(* IEC 61131-3 sources: B-R/MBA, 12 files *)

(* ---- Main.st ---- *)
PROGRAM _INIT
	(* Insert code here *)
	MBAPid0510Para.set_value := 25;
	MBAPid0802Para.set_value := 30;
	MBAPid0510Para.gain := 400;
	MBAPid0802Para.gain := 60;
	MBAPid0510Para.integration_time := 45;
	MBAPid0802Para.integration_time := 240;
	MBAPid0510Para.derivative_time := 30;
	MBAPid0802Para.derivative_time := 0;

END_PROGRAM

PROGRAM _CYCLIC
	(* Insert code here *)
	S1A_ACT;
	S1B_ACT;
	S2_ACT;
	S3_ACT;
	S4_ACT;
	S5_ACT;
	S6_ACT;
	S7_ACT;
	S8_ACT;
	S9_ACT;
	S10_ACT;
END_PROGRAM

(* ---- MBAS10_ACTION.st ---- *)
ACTION S10_ACT:
	//设定时间
	FOR i := 0 TO MBAS10_STEP_NUM DO
		IF MBAS10_ST[i] < T#5s THEN
			MBAS10_ST[i] := T#5s;
		END_IF;
		MBAS10_STEP[i].set_time := MBAS10_ST[i];
	END_FOR;

	//流程步骤
	ProcessHandleFC(MBAS10,MBAS10_STEP[0],MBAS10_STEP_NUM);

	//object 手自动切换
	IF (MBAS10.status.mode <> 0) AND (NOT MBAS10.auto_mode_edge) THEN
		MBAS10.auto_mode_edge := TRUE;
		MBAS10.manual_mode_edge := FALSE;

		MBAR11.control.auto_operate := TRUE;
		MBAXV0811.control.auto_operate := TRUE;
		MBAXV0807.control.auto_operate := TRUE;
		MBAXV0808.control.auto_operate := TRUE;
		MBAXV0809.control.auto_operate := TRUE;
		MBAP09.control.auto_operate := TRUE;
		MBATV0801A.control.auto_operate := TRUE;
		MBATV0801B.control.auto_operate := TRUE;
		MBAXV0806.control.auto_operate := TRUE;
		MBAXV0812.control.auto_operate := TRUE;
		MBATVT0802.control.auto_operate := TRUE;
	END_IF;

	IF (MBAS10.status.mode = 0) AND (NOT MBAS10.manual_mode_edge) THEN
		MBAS10.manual_mode_edge := TRUE;
		MBAS10.auto_mode_edge := FALSE;

		MBAR11.control.manual_operate := TRUE;
		MBAXV0811.control.manual_operate := TRUE;
		MBAXV0807.control.manual_operate := TRUE;
		MBAXV0808.control.manual_operate := TRUE;
		MBAXV0809.control.manual_operate := TRUE;
		MBAP09.control.manual_operate := TRUE;
		MBATV0801A.control.manual_operate := TRUE;
		MBATV0801B.control.manual_operate := TRUE;
		MBAXV0806.control.manual_operate := TRUE;
		MBAXV0812.control.manual_operate := TRUE;
		MBATVT0802.control.manual_operate := TRUE;
	END_IF;

	//错误信号停机
	MBAS10.input.error_signal := (MBAR11.status.motor_status >= 2) OR (MBAXV0811.status.valve_status >= 2) OR
	(MBAXV0807.status.valve_status >= 2) OR (MBAXV0808.status.valve_status >= 2) OR (MBAXV0809.status.valve_status >= 2) OR
	(MBAP09.status.motor_status >= 2) OR (MBATV0801A.status.valve_status >= 2) OR (MBATV0801B.status.valve_status >= 2) OR
	(MBAXV0806.status.valve_status >= 2) OR (MBAXV0812.status.valve_status >= 2) OR (MBATVT0802.status.regulator_status >= 2);

	//MBAXV0814 玻璃塔出料自动
	SquareWave_0(open_time := DINT_TO_TIME(MBAXV0814_Open_Time * 1000), close_time := DINT_TO_TIME(MBAXV0814_Close_Time * 1000), on_off := TRUE, out := MBAXV0814.input.auto_open_signal);
	IF MBAS10.status.run_state = 1 THEN
		//步骤执行动作
		CASE MBAS10.status.run_step OF
			0:
				MBAS10_STEP[0].done := TRUE;
			1:
				//人工加料
			2:
				MBAR11.input.auto_run_signal := TRUE;
				MBAXV0811.input.auto_open_signal := TRUE;
				MBAXV0807.input.auto_open_signal := TRUE;
				MBAXV0808.input.auto_open_signal := TRUE;
				MBAXV0809.input.auto_open_signal := TRUE;
				MBAP09.input.auto_run_signal := TRUE;
				MTBasicsPID_1.Enable := TRUE;
				MBAS10_STEP[2].done := TRUE;
			3:
				IF (MBATIT0801.status.value < MBAS10_PARA_Temp1) AND (NOT MBAS10_STEP[3].done) THEN
	 				MBATV0801A.input.auto_open_signal := TRUE;
				END_IF;
				IF MBATIT0801.status.value >= MBAS10_PARA_Temp1 THEN
					MBATV0801B.input.auto_open_signal := TRUE;
					MBATV0801A.input.auto_open_signal := FALSE;
					MBAS10_STEP[3].done := TRUE;
				END_IF;
			4:

			5:
				IF MBATIT0803.status.value >= MBAS10_PARA_Temp2 THEN
					MBAXV0806.input.auto_open_signal := TRUE;
					MBAXV0807.input.auto_open_signal := FALSE;
					MBAXV0808.input.auto_open_signal := FALSE;
					MBAS10_STEP[5].done := TRUE;
				END_IF;
			6:
				IF MBATIT0801.status.value >= MBAS10_PARA_Temp3 THEN
					MBATV0801B.input.auto_open_signal := FALSE;
					MBAXV0807.input.auto_open_signal := TRUE;
					MBAXV0808.input.auto_open_signal := TRUE;
					MBAXV0806.input.auto_open_signal := FALSE;
					MBAXV0809.input.auto_open_signal := FALSE;
					MBAS10_STEP[6].done := TRUE;
				END_IF;
			7:
				IF MBATIT0801.status.value <= MBAS10_PARA_Temp4 THEN
					MBAXV0807.input.auto_open_signal := FALSE;
					MBAXV0808.input.auto_open_signal := FALSE;
					MBAXV0812.input.auto_open_signal := TRUE;
					MBAP09.input.auto_run_signal := FALSE;
					MBAS10_STEP[7].done := TRUE;
				END_IF;
			8:
			//人工操作
		END_CASE;
	END_IF;

	//TSV0510调节
	R_TRIG_3(CLK := MBATVT0802.status.auto_mode);
	IF R_TRIG_3.Q THEN
		MTBasicsPID_1.Enable := TRUE;
	END_IF;
	F_TRIG_3(CLK := MBATVT0802.status.auto_mode);
	IF F_TRIG_3.Q THEN
		MTBasicsPID_1.Enable := FALSE;
	END_IF;
	//MTBasicsPID_1.Enable := TRUE;
	MTBasicsPID_1.Invert := TRUE;
	MTBasicsPID_1.PIDParameters.Gain := MBAPid0802Para.gain;
	MTBasicsPID_1.PIDParameters.DerivativeTime := MBAPid0802Para.derivative_time;
	MTBasicsPID_1.PIDParameters.IntegrationTime := MBAPid0802Para.integration_time;
	MTBasicsPID_1.MinOut := 0.0;
	MTBasicsPID_1.MaxOut := 100.0;
	MTBasicsPID_1.SetValue := MBAPid0802Para.set_value;
	MTBasicsPID_1.ActValue := MBATIT0802.status.value;
	MTBasicsPID_1.Update := MBAPid0802.update;
	MTBasicsPID_1();
	MBAPid0802.out := MTBasicsPID_1.Out;
	IF MTBasicsPID_1.Active THEN
		MBATVT0802.input.auto_degree_set := MTBasicsPID_1.Out;
	ELSE
		MBATVT0802.input.auto_degree_set := 0.0;
	END_IF;
	IF MTBasicsPID_1.UpdateDone THEN
		MBAPid0802.update := FALSE;
	END_IF;

	//人工确认步骤可用
	IF (MBAS10.status.run_state) AND (NOT MBAS10_STEP[MBAS10.status.run_step].done AND ((MBAS10.status.run_step = 1) OR (MBAS10.status.run_step = 4) OR (MBAS10.status.run_step = 8))) THEN
		MBAS10.status.confirm_enable := TRUE;
	ELSE
		MBAS10.status.confirm_enable := FALSE;
	END_IF;
END_ACTION

(* ---- MBAS1A_ACTION.st ---- *)
ACTION S1A_ACT:
	//设定时间
	FOR i := 0 TO MBAS1_STEP_NUM DO
		IF MBAS1A_ST[i] < T#5s THEN
			MBAS1A_ST[i] := T#5s;
		END_IF;
		MBAS1A_STEP[i].set_time := MBAS1A_ST[i];
	END_FOR;

	//流程步骤
	ProcessHandleFC(MBAS1A,MBAS1A_STEP[0],MBAS1_STEP_NUM);

	//object 手自动切换
	IF (MBAS1A.status.mode <> 0) AND (NOT MBAS1A.auto_mode_edge) THEN
		MBAS1A.auto_mode_edge := TRUE;
		MBAS1A.manual_mode_edge := FALSE;

		STFLV0101.control.auto_operate := TRUE;
		STFLV0102.control.auto_operate := TRUE;
		MBALV0102.control.auto_operate := TRUE;
		STFP01.control.auto_operate := TRUE;
		STFLV3601.control.auto_operate := TRUE;
		STFLV3602.control.auto_operate := TRUE;
		MBALV0103.control.auto_operate := TRUE;
		STFP36.control.auto_operate := TRUE;
		MBALV0101.control.auto_operate := TRUE;
		MBAXV0105.control.auto_operate := TRUE;
		MBAXV0103.control.auto_operate := TRUE;
		MBAAV0101A.control.auto_operate := TRUE;
		MBAR01A.control.auto_operate := TRUE;
		MBAXV0102.control.auto_operate := TRUE;
		MBAXV0101.control.auto_operate := TRUE;
		MBAAV0101B.control.auto_operate := TRUE;
		MBAXV0209.control.auto_operate := TRUE;
		MBAXV0212.control.auto_operate := TRUE;
		MBAXV0104.control.auto_operate := TRUE;
		MBAXV0415.control.auto_operate := TRUE;
	END_IF;

	IF (MBAS1A.status.mode = 0) AND (NOT MBAS1A.manual_mode_edge) THEN
		MBAS1A.manual_mode_edge := TRUE;
		MBAS1A.auto_mode_edge := FALSE;

		STFLV0101.control.manual_operate := TRUE;
		STFLV0102.control.manual_operate := TRUE;
		MBALV0102.control.manual_operate := TRUE;
		STFP01.control.manual_operate := TRUE;
		STFLV3601.control.manual_operate := TRUE;
		STFLV3602.control.manual_operate := TRUE;
		MBALV0103.control.manual_operate := TRUE;
		STFP36.control.manual_operate := TRUE;
		MBALV0101.control.manual_operate := TRUE;
		MBAXV0105.control.manual_operate := TRUE;
		MBAXV0103.control.manual_operate := TRUE;
		MBAAV0101A.control.manual_operate := TRUE;
		MBAR01A.control.manual_operate := TRUE;
		MBAXV0102.control.manual_operate := TRUE;
		MBAXV0101.control.manual_operate := TRUE;
		MBAAV0101B.control.manual_operate := TRUE;
		MBAXV0209.control.manual_operate := TRUE;
		MBAXV0212.control.manual_operate := TRUE;
		MBAXV0104.control.manual_operate := TRUE;
		MBAXV0415.control.manual_operate := TRUE;
	END_IF;

	//错误信号停机
	MBAS1A.input.error_signal := (STFLV0101.status.valve_status >= 2) OR (STFLV0102.status.valve_status >= 2) OR
	(MBALV0102.status.valve_status >= 2) OR (STFP01.status.motor_status >= 2) OR (STFLV3601.status.valve_status >= 2) OR
	(STFLV3602.status.valve_status >= 2) OR (MBALV0103.status.valve_status >= 2) OR (STFP36.status.motor_status >= 2) OR
	(MBALV0101.status.valve_status >= 2) OR (MBAXV0105.status.valve_status >= 2) OR (MBAXV0103.status.valve_status >= 2) OR
	(MBAAV0101A.status.valve_status >= 2) OR (MBAR01A.status.motor_status >= 2) OR (MBAXV0102.status.valve_status >= 2) OR
	(MBAXV0101.status.valve_status >= 2) OR (MBAAV0101B.status.valve_status >= 2) OR (MBAXV0209.status.valve_status >= 2) OR
	(MBAXV0212.status.valve_status >= 2) OR (MBAXV0104.status.valve_status >= 2) OR (MBAXV0415.status.valve_status >= 2);

	IF MBAS1A.status.run_state = 1 THEN
		//步骤执行动作
		CASE MBAS1A.status.run_step OF
			0:
				IF NOT MBAS1A_STEP[0].done  THEN
					STFLV0101.control.auto_operate := TRUE;
					STFLV0102.control.auto_operate := TRUE;
					MBALV0104.control.auto_operate := TRUE;
					STFP01.control.auto_operate := TRUE;
					STFLV3601.control.auto_operate := TRUE;
					STFLV3602.control.auto_operate := TRUE;
					MBALV0105.control.auto_operate := TRUE;
					STFP36.control.auto_operate := TRUE;
					MBALV0101.control.auto_operate := TRUE;
					MBAXV0110.control.auto_operate := TRUE;
					MBAXV0108.control.auto_operate := TRUE;
					MBAAV0102A.control.auto_operate := TRUE;
					MBAR01B.control.auto_operate := TRUE;
					MBAXV0107.control.auto_operate := TRUE;
					MBAXV0106.control.auto_operate := TRUE;
					MBAAV0102B.control.auto_operate := TRUE;
					MBAXV0209.control.auto_operate := TRUE;
					MBAXV0212.control.auto_operate := TRUE;
					MBAXV0109.control.auto_operate := TRUE;
					MBAXV0415.control.auto_operate := TRUE;
					MBAS1A_STEP[0].done := TRUE;
				END_IF;
			1:
				//高位槽进料
			2:
				CASE step1_4a OF
					0:
						IF NOT MBAS1A_STEP[2].done THEN
							step1_4a := 1;
						END_IF;
					1:
						MBAXV0105.input.auto_open_signal := TRUE;
						step1_4a := 2;
					2:
						TON_8.PT := DINT_TO_TIME(MBAS1A_PARA_T4 * 1000);
						TON_8.IN := TRUE;
						IF TON_8.Q THEN
							TON_8.IN := FALSE;
							step1_4a := 3;
						END_IF;
					3:
						MBAXV0105.input.auto_open_signal := FALSE;
						step1_4a := 4;
					4:
						MBAXV0103.input.auto_open_signal := TRUE;
						IF MBAXV0103.input.open_feedback_state THEN
							step1_4a := 5;
						END_IF;
					5:
						IF MBALIT0101.status.value <= MBAS1A_PARA_L4 THEN
							step1_4a := 6;
						END_IF;
					6:
						TON_8.PT := DINT_TO_TIME(MBAS1A_PARA_T5 * 60 * 1000);
						TON_8.IN := TRUE;
						IF TON_8.Q THEN
							TON_8.IN := FALSE;
							step1_4a := 7;
						END_IF;
					7:
						MBAXV0103.input.auto_open_signal := FALSE;
						IF MBAXV0103.input.close_feedback_state THEN
							step1_4a := 0;
							MBAS1A_STEP[2].done := TRUE;
						END_IF;
				END_CASE;
				TON_8();
			3:
				//人工投料,结束后确认
			4:
				CASE step1_6a OF
					0:
						IF NOT MBAS1A_STEP[4].done THEN
							step1_6a := 1;
						END_IF;
					1:
						LiquidRelease_3(sp_time := DINT_TO_TIME(MBAS1A_PARA_T10 * 60 * 1000),
						level_value := MBALIT0102.status.value,
						set_point := MBAS1A_PARA_L5,
						done := step1_6a_1_done);
						MBAAV0101A.input.auto_open_signal := LiquidRelease_3.run;
						IF step1_6a_1_done AND MBAAV0101A.input.close_feedback_state AND (NOT MBAAV0101A.input.auto_open_signal) THEN
							step1_6a := 2;
						END_IF;
					2:
						MBAR01A.input.auto_run_signal := TRUE;
						IF MBAR01A.input.run_feedback THEN
							step1_6a := 0;
							step1_6a_1_done := FALSE;
							MBAS1A_STEP[4].done := TRUE;
						END_IF;
				END_CASE;
			5:
				CASE step1_7a OF
					0:
						IF NOT MBAS1A_STEP[5].done THEN
							step1_7a := 1;
						END_IF;
					1:
						TON_13.PT := DINT_TO_TIME(MBAS1A_PARA_T6 * 60 * 1000);
						TON_13.IN := TRUE;
						IF TON_13.Q THEN
							TON_13.IN := FALSE;
							step1_7a := 2;
						END_IF;
					2:
						MBAXV0101.input.auto_open_signal := TRUE;
						IF MBAXV0101.input.open_feedback_state THEN
							step1_7a := 3;
						END_IF;
					3:
						IF MBATIT0101.status.value >= MBAS1A_PARA_Temp1 THEN
							step1_7a := 4;
						END_IF;
					4:
						MBAXV0102.input.auto_open_signal := TRUE;
						IF MBAXV0102.input.open_feedback_state THEN
							step1_7a := 5;
						END_IF;
					5:
						TON_13.PT := DINT_TO_TIME(MBAS1A_PARA_T7 * 60 * 1000);
						TON_13.IN := TRUE;
						IF TON_13.Q THEN
							TON_13.IN := FALSE;
							step1_7a := 6;
						END_IF;
					6:
						MBAAV0101B.input.auto_open_signal := TRUE;
						IF MBAAV0101B.input.open_feedback_state THEN
							step1_7a := 7;
						END_IF;
					7:
						TON_13.PT := DINT_TO_TIME(MBAS1A_PARA_T8 * 60 * 1000);
						TON_13.IN := TRUE;
						IF TON_13.Q THEN
							TON_13.IN := FALSE;
							step1_7a := 8;
						END_IF;
					8:
						MBAAV0101A.input.auto_open_signal := TRUE;
						IF MBAAV0101A.input.open_feedback_state THEN
							step1_7a := 9;
						END_IF;
					9:
						TON_13.PT := DINT_TO_TIME(MBAS1A_PARA_T9 * 60 * 1000);
						TON_13.IN := TRUE;
						IF TON_13.Q THEN
							TON_13.IN := FALSE;
							step1_7a := 10;
						END_IF;
					10:
						MBAXV0102.input.auto_open_signal := FALSE;
						MBAAV0101A.input.auto_open_signal := FALSE;
						MBAAV0101B.input.auto_open_signal := FALSE;
						IF MBAXV0102.input.close_feedback_state AND MBAAV0101A.input.close_feedback_state AND MBAAV0101B.input.close_feedback_state THEN
							step1_7a := 0;
							MBAS1A_STEP[5].done := TRUE;
						END_IF;
				END_CASE;
				TON_13();
			6:
				//人工确认MBAR13空闲
			7:
				MBAXV0209.input.auto_open_signal := TRUE;
				MBAXV0212.input.auto_open_signal := TRUE;
				MBAXV0415.input.auto_open_signal := TRUE;
				IF MBAXV0209.input.open_feedback_state AND MBAXV0212.input.open_feedback_state AND MBAXV0415.input.open_feedback_state THEN
					MBAXV0104.input.auto_open_signal := TRUE;
					MBAR01A.input.auto_run_signal := FALSE;
				END_IF;
				IF MBAXV0209.input.open_feedback_state AND MBAXV0212.input.open_feedback_state AND MBAXV0415.input.open_feedback_state AND MBAXV0104.input.open_feedback_state AND (NOT MBAR01A.input.run_feedback) THEN
					MBAS1A_STEP[7].done := TRUE;
				END_IF;
			8:
				//人工确认转移完毕
			9:
				MBAXV0104.input.auto_open_signal := FALSE;
				MBAXV0101.input.auto_open_signal := FALSE;
				IF MBAXV0104.input.close_feedback_state AND MBAXV0101.input.close_feedback_state THEN
					MBAS1A_STEP[9].done := TRUE;
				END_IF;
		END_CASE;
	END_IF;

	IF mba_v02a_add THEN
		CASE step1_1a OF
			0:
				step1_1a := 1;
			1:
				STFLV0101.input.auto_open_signal := FALSE;
				STFLV0102.input.auto_open_signal := FALSE;
				MBALV0102.input.auto_open_signal := TRUE;
				IF STFLV0102.input.close_feedback_state AND STFLV0101.input.close_feedback_state AND MBALV0102.input.open_feedback_state THEN
					step1_1a := 2;
				END_IF;
			2:
				LiquidAdd_0(level_value := MBALIT0102.status.value,
				sp_value := MBAS1A_PARA_L1,
				sp_accumulation := MBAS1A_PARA_AC1,
				sp_time := DINT_TO_TIME(MBAS1A_PARA_T1 * 1000),
				flowmeter := STFFQIT0102,
				done := step1_1a_2_done);
				STFP01.input.auto_run_signal := LiquidAdd_0.run;
				IF step1_1a_2_done AND (NOT STFP01.input.run_feedback) AND (NOT STFP01.input.auto_run_signal) THEN
					step1_1a := 3;
				END_IF;
			3:
				IF STFFQIT0102.flowrate <= flowrate_threshold THEN
					step1_1a := 4;
				END_IF;
			4:
				MBALV0102.input.auto_open_signal := FALSE;
				IF MBALV0102.input.close_feedback_state THEN
					step1_1a_2_done := FALSE;
					step1_1a := 0;
					mba_v02a_add := FALSE;
				END_IF;
		END_CASE;
	END_IF;

	IF mba_v03a_add THEN
		CASE step1_2a OF
			0:
				step1_2a := 1;
			1:
				STFLV3601.input.auto_open_signal := TRUE;
				STFLV3602.input.auto_open_signal := FALSE;
				MBALV0103.input.auto_open_signal := TRUE;
				IF STFLV3601.input.open_feedback_state AND STFLV3602.input.close_feedback_state AND MBALV0103.input.open_feedback_state THEN
					step1_2a := 2;
				END_IF;
			2:
				LiquidAdd_1(level_value := MBALIT0103.status.value,
				sp_value := MBAS1A_PARA_L2,
				sp_accumulation := MBAS1A_PARA_AC2,
				sp_time := DINT_TO_TIME(MBAS1A_PARA_T2 * 1000),
				flowmeter := STFFQIT3602,
				done := step1_2a_2_done);
				STFP36.input.auto_run_signal := LiquidAdd_1.run;
				IF step1_2a_2_done AND (NOT STFP36.input.run_feedback) AND (NOT STFP36.input.auto_run_signal) THEN
					step1_2a := 3;
				END_IF;
			3:
				IF STFFQIT3602.flowrate <= flowrate_threshold THEN
					step1_2a := 4;
				END_IF;
			4:
				MBALV0103.input.auto_open_signal := FALSE;
				IF MBALV0103.input.close_feedback_state THEN
					step1_2a := 0;
					step1_2a_2_done := FALSE;
					mba_v03a_add := FALSE;
				END_IF;
		END_CASE;
	END_IF;

	//人工确认步骤可用
	IF (MBAS1A.status.run_state) AND (NOT MBAS1A_STEP[MBAS1A.status.run_step].done AND ((MBAS1A.status.run_step = 1) OR (MBAS1A.status.run_step = 3) OR (MBAS1A.status.run_step = 6) OR (MBAS1A.status.run_step = 8))) THEN
		MBAS1A.status.confirm_enable := TRUE;
	ELSE
		MBAS1A.status.confirm_enable := FALSE;
	END_IF;
END_ACTION

(* ---- MBAS1B_ACTION.st ---- *)
ACTION S1B_ACT:
	//设定时间
	FOR i := 0 TO MBAS1_STEP_NUM DO
		IF MBAS1B_ST[i] < T#5s THEN
			MBAS1B_ST[i] := T#5s;
		END_IF;
		MBAS1B_STEP[i].set_time := MBAS1B_ST[i];
	END_FOR;

	//流程步骤
	ProcessHandleFC(MBAS1B,MBAS1B_STEP[0],MBAS1_STEP_NUM);

	//object 手自动切换
	IF (MBAS1B.status.mode <> 0) AND (NOT MBAS1B.auto_mode_edge) THEN
		MBAS1B.auto_mode_edge := TRUE;
		MBAS1B.manual_mode_edge := FALSE;

		STFLV0101.control.auto_operate := TRUE;
		STFLV0102.control.auto_operate := TRUE;
		MBALV0104.control.auto_operate := TRUE;
		STFP01.control.auto_operate := TRUE;
		STFLV3601.control.auto_operate := TRUE;
		STFLV3602.control.auto_operate := TRUE;
		MBALV0105.control.auto_operate := TRUE;
		STFP36.control.auto_operate := TRUE;
		MBALV0101.control.auto_operate := TRUE;
		MBAXV0110.control.auto_operate := TRUE;
		MBAXV0108.control.auto_operate := TRUE;
		MBAAV0102A.control.auto_operate := TRUE;
		MBAR01B.control.auto_operate := TRUE;
		MBAXV0107.control.auto_operate := TRUE;
		MBAXV0106.control.auto_operate := TRUE;
		MBAAV0102B.control.auto_operate := TRUE;
		MBAXV0209.control.auto_operate := TRUE;
		MBAXV0212.control.auto_operate := TRUE;
		MBAXV0109.control.auto_operate := TRUE;
		MBAXV0415.control.auto_operate := TRUE;
	END_IF;

	IF (MBAS1B.status.mode = 0) AND (NOT MBAS1B.manual_mode_edge) THEN
		MBAS1B.manual_mode_edge := TRUE;
		MBAS1B.auto_mode_edge := FALSE;

		STFLV0101.control.manual_operate := TRUE;
		STFLV0102.control.manual_operate := TRUE;
		MBALV0104.control.manual_operate := TRUE;
		STFP01.control.manual_operate := TRUE;
		STFLV3601.control.manual_operate := TRUE;
		STFLV3602.control.manual_operate := TRUE;
		MBALV0105.control.manual_operate := TRUE;
		STFP36.control.manual_operate := TRUE;
		MBALV0101.control.manual_operate := TRUE;
		MBAXV0110.control.manual_operate := TRUE;
		MBAXV0108.control.manual_operate := TRUE;
		MBAAV0102A.control.manual_operate := TRUE;
		MBAR01B.control.manual_operate := TRUE;
		MBAXV0107.control.manual_operate := TRUE;
		MBAXV0106.control.manual_operate := TRUE;
		MBAAV0102B.control.manual_operate := TRUE;
		MBAXV0209.control.manual_operate := TRUE;
		MBAXV0212.control.manual_operate := TRUE;
		MBAXV0109.control.manual_operate := TRUE;
		MBAXV0415.control.manual_operate := TRUE;
	END_IF;

	//错误信号停机
	MBAS1B.input.error_signal := (STFLV0101.status.valve_status >= 2) OR (STFLV0102.status.valve_status >= 2) OR
	(MBALV0104.status.valve_status >= 2) OR (STFP01.status.motor_status >= 2) OR (STFLV3601.status.valve_status >= 2) OR
	(STFLV3602.status.valve_status >= 2) OR (MBALV0105.status.valve_status >= 2) OR (STFP36.status.motor_status >= 2) OR
	(MBALV0101.status.valve_status >= 2) OR (MBAXV0110.status.valve_status >= 2) OR (MBAXV0108.status.valve_status >= 2) OR
	(MBAAV0102A.status.valve_status >= 2) OR (MBAR01B.status.motor_status >= 2) OR (MBAXV0107.status.valve_status >= 2) OR
	(MBAXV0106.status.valve_status >= 2) OR (MBAAV0102B.status.valve_status >= 2) OR (MBAXV0209.status.valve_status >= 2) OR
	(MBAXV0212.status.valve_status >= 2) OR (MBAXV0109.status.valve_status >= 2) OR (MBAXV0415.status.valve_status >= 2);

	IF MBAS1B.status.run_state = 1 THEN
		//步骤执行动作
		CASE MBAS1B.status.run_step OF
			0:
				IF NOT MBAS1B_STEP[0].done THEN
					STFLV0101.control.auto_operate := TRUE;
					STFLV0102.control.auto_operate := TRUE;
					MBALV0104.control.auto_operate := TRUE;
					STFP01.control.auto_operate := TRUE;
					STFLV3601.control.auto_operate := TRUE;
					STFLV3602.control.auto_operate := TRUE;
					MBALV0105.control.auto_operate := TRUE;
					STFP36.control.auto_operate := TRUE;
					MBALV0101.control.auto_operate := TRUE;
					MBAXV0110.control.auto_operate := TRUE;
					MBAXV0108.control.auto_operate := TRUE;
					MBAAV0102A.control.auto_operate := TRUE;
					MBAR01B.control.auto_operate := TRUE;
					MBAXV0107.control.auto_operate := TRUE;
					MBAXV0106.control.auto_operate := TRUE;
					MBAAV0102B.control.auto_operate := TRUE;
					MBAXV0209.control.auto_operate := TRUE;
					MBAXV0212.control.auto_operate := TRUE;
					MBAXV0109.control.auto_operate := TRUE;
					MBAXV0415.control.auto_operate := TRUE;
					MBAS1B_STEP[0].done := TRUE;
				END_IF;
			1:
				//高位槽进料
			2:
				CASE step1_4b OF
					0:
						IF NOT MBAS1B_STEP[2].done THEN
							step1_4b := 1;
						END_IF;
					1:
						MBAXV0110.input.auto_open_signal := TRUE;
						step1_4b := 2;
					2:
						TON_14.PT := DINT_TO_TIME(MBAS1B_PARA_T4 * 1000);
						TON_14.IN := TRUE;
						IF TON_14.Q THEN
							TON_14.IN := FALSE;
							step1_4b := 3;
						END_IF;
					3:
						MBAXV0110.input.auto_open_signal := FALSE;
						step1_4b := 4;
					4:
						MBAXV0108.input.auto_open_signal := TRUE;
						IF MBAXV0108.input.open_feedback_state THEN
							step1_4b := 5;
						END_IF;
					5:
						IF MBALIT0101.status.value <= MBAS1B_PARA_L4 THEN
							step1_4b := 6;
						END_IF;
					6:
						TON_14.PT := DINT_TO_TIME(MBAS1B_PARA_T5 * 60 * 1000);
						TON_14.IN := TRUE;
						IF TON_14.Q THEN
							TON_14.IN := FALSE;
							step1_4b := 7;
						END_IF;
					7:
						MBAXV0108.input.auto_open_signal := FALSE;
						IF MBAXV0108.input.close_feedback_state THEN
							step1_4b := 0;
							MBAS1B_STEP[2].done := TRUE;
						END_IF;
				END_CASE;
				TON_14();
			3:
				//人工投料,结束后确认
			4:
				CASE step1_6b OF
					0:
						IF NOT MBAS1B_STEP[4].done THEN
							step1_6b := 1;
						END_IF;
					1:
						LiquidRelease_1(sp_time := DINT_TO_TIME(MBAS1B_PARA_T10 * 60 * 1000),
						level_value := MBALIT0104.status.value,
						set_point := MBAS1B_PARA_L5,
						done := step1_6b_1_done);
						MBAAV0102A.input.auto_open_signal := LiquidRelease_1.run;
						IF step1_6b_1_done AND MBAAV0102A.input.close_feedback_state AND (NOT MBAAV0102A.input.auto_open_signal) THEN
							step1_6b := 2;
						END_IF;
					2:
						MBAR01B.input.auto_run_signal := TRUE;
						IF MBAR01B.input.run_feedback THEN
							step1_6b := 0;
							step1_6b_1_done := FALSE;
							MBAS1B_STEP[4].done := TRUE;
						END_IF;
				END_CASE;
			5:
				CASE step1_7b OF
					0:
						IF NOT MBAS1B_STEP[5].done THEN
							step1_7b := 1;
						END_IF;
					1:
						TON_15.PT := DINT_TO_TIME(MBAS1B_PARA_T6 * 60 * 1000);
						TON_15.IN := TRUE;
						IF TON_15.Q THEN
							TON_15.IN := FALSE;
							step1_7b := 2;
						END_IF;
					2:
						MBAXV0106.input.auto_open_signal := TRUE;
						IF MBAXV0106.input.open_feedback_state THEN
							step1_7b := 3;
						END_IF;
					3:
						IF MBATIT0102.status.value >= MBAS1B_PARA_Temp1 THEN
							step1_7b := 4;
						END_IF;
					4:
						MBAXV0107.input.auto_open_signal := TRUE;
						IF MBAXV0107.input.open_feedback_state THEN
							step1_7b := 5;
						END_IF;
					5:
						TON_15.PT := DINT_TO_TIME(MBAS1B_PARA_T7 * 60 * 1000);
						TON_15.IN := TRUE;
						IF TON_15.Q THEN
							TON_15.IN := FALSE;
							step1_7b := 6;
						END_IF;
					6:
						MBAAV0102B.input.auto_open_signal := TRUE;
						IF MBAAV0102B.input.open_feedback_state THEN
							step1_7b := 7;
						END_IF;
					7:
						TON_15.PT := DINT_TO_TIME(MBAS1B_PARA_T8 * 60 * 1000);
						TON_15.IN := TRUE;
						IF TON_15.Q THEN
							TON_15.IN := FALSE;
							step1_7b := 8;
						END_IF;
					8:
						MBAAV0102A.input.auto_open_signal := TRUE;
						IF MBAAV0102A.input.open_feedback_state THEN
							step1_7b := 9;
						END_IF;
					9:
						TON_15.PT := DINT_TO_TIME(MBAS1B_PARA_T9 * 60 * 1000);
						TON_15.IN := TRUE;
						IF TON_15.Q THEN
							TON_15.IN := FALSE;
							step1_7b := 10;
						END_IF;
					10:
						MBAXV0107.input.auto_open_signal := FALSE;
						MBAAV0102A.input.auto_open_signal := FALSE;
						MBAAV0102B.input.auto_open_signal := FALSE;
						IF MBAXV0107.input.close_feedback_state AND MBAAV0102A.input.close_feedback_state AND MBAAV0102B.input.close_feedback_state THEN
							step1_7b := 0;
							MBAS1B_STEP[5].done := TRUE;
						END_IF;
				END_CASE;
				TON_15();
			6:
				//人工确认MBAR13空闲
			7:
				MBAXV0209.input.auto_open_signal := TRUE;
				MBAXV0212.input.auto_open_signal := TRUE;
				MBAXV0415.input.auto_open_signal := TRUE;
				IF MBAXV0209.input.open_feedback_state AND MBAXV0212.input.open_feedback_state AND MBAXV0415.input.open_feedback_state THEN
					MBAXV0109.input.auto_open_signal := TRUE;
					MBAR01B.input.auto_run_signal := FALSE;
				END_IF;
				IF MBAXV0209.input.open_feedback_state AND MBAXV0212.input.open_feedback_state AND MBAXV0415.input.open_feedback_state AND MBAXV0109.input.open_feedback_state AND (NOT MBAR01B.input.run_feedback) THEN
					MBAS1B_STEP[7].done := TRUE;
				END_IF;
			8:
				//人工确认转移完毕
			9:
				MBAXV0109.input.auto_open_signal := FALSE;
				MBAXV0106.input.auto_open_signal := FALSE;
				IF MBAXV0109.input.close_feedback_state AND MBAXV0106.input.close_feedback_state THEN
					MBAS1B_STEP[9].done := TRUE;
				END_IF;
		END_CASE;
	END_IF;

	IF mba_v02b_add THEN
		CASE step1_1b OF
			0:
				step1_1b := 1;
			1:
				STFLV0101.input.auto_open_signal := FALSE;
				STFLV0102.input.auto_open_signal := FALSE;
				MBALV0104.input.auto_open_signal := TRUE;
				IF STFLV0102.input.close_feedback_state AND STFLV0101.input.close_feedback_state AND MBALV0104.input.open_feedback_state THEN
					step1_1b := 2;
				END_IF;
			2:
				LiquidAdd_4(level_value := MBALIT0104.status.value,
				sp_value := MBAS1B_PARA_L1,
				sp_accumulation := MBAS1B_PARA_AC1,
				sp_time := DINT_TO_TIME(MBAS1B_PARA_T1 * 1000),
				flowmeter := STFFQIT0102,
				done := step1_1b_2_done);
				STFP01.input.auto_run_signal := LiquidAdd_4.run;
				IF step1_1b_2_done AND (NOT STFP01.input.run_feedback) AND (NOT STFP01.input.auto_run_signal) THEN
					step1_1b := 3;
				END_IF;
			3:
				IF STFFQIT0102.flowrate <= flowrate_threshold THEN
					step1_1b := 4;
				END_IF;
			4:
				MBALV0104.input.auto_open_signal := FALSE;
				IF MBALV0104.input.close_feedback_state THEN
					step1_1b := 0;
					step1_1b_2_done := FALSE;
					mba_v02b_add := FALSE;
				END_IF;
		END_CASE;
	END_IF;

	IF mba_v03b_add THEN
		CASE step1_2b OF
			0:
				step1_2b := 1;
			1:
				STFLV3601.input.auto_open_signal := TRUE;
				STFLV3602.input.auto_open_signal := FALSE;
				MBALV0105.input.auto_open_signal := TRUE;
				IF STFLV3601.input.open_feedback_state AND STFLV3602.input.close_feedback_state AND MBALV0105.input.open_feedback_state THEN
					step1_2b := 2;
				END_IF;
			2:
				LiquidAdd_5(level_value := MBALIT0105.status.value,
				sp_value := MBAS1B_PARA_L2,
				sp_accumulation := MBAS1B_PARA_AC2,
				sp_time := DINT_TO_TIME(MBAS1B_PARA_T2 * 1000),
				flowmeter := STFFQIT3602,
				done := step1_2b_2_done);
				STFP36.input.auto_run_signal := LiquidAdd_5.run;
				IF step1_2b_2_done AND (NOT STFP36.input.run_feedback) AND (NOT STFP36.input.auto_run_signal) THEN
					step1_2b := 3;
				END_IF;
			3:
				IF STFFQIT3602.flowrate <= flowrate_threshold THEN
					step1_2b := 4;
				END_IF;
			4:
				MBALV0105.input.auto_open_signal := FALSE;
				IF MBALV0105.input.close_feedback_state THEN
					step1_2b := 0;
					step1_2b_2_done := FALSE;
					mba_v03b_add := FALSE;
				END_IF;
		END_CASE;
	END_IF;

	//人工确认步骤可用
	IF (MBAS1B.status.run_state) AND (NOT MBAS1B_STEP[MBAS1B.status.run_step].done AND ((MBAS1B.status.run_step = 1) OR (MBAS1B.status.run_step = 3) OR (MBAS1B.status.run_step = 6) OR (MBAS1B.status.run_step = 8))) THEN
		MBAS1B.status.confirm_enable := TRUE;
	ELSE
		MBAS1B.status.confirm_enable := FALSE;
	END_IF;
END_ACTION

(* ---- MBAS2_ACTION.st ---- *)
ACTION S2_ACT:
	//设定时间
	FOR i := 0 TO MBAS2_STEP_NUM DO
		IF MBAS2_ST[i] < T#5s THEN
			MBAS2_ST[i] := T#5s;
		END_IF;
		MBAS2_STEP[i].set_time := MBAS2_ST[i];
	END_FOR;

	//流程步骤
	ProcessHandleFC(MBAS2,MBAS2_STEP[0],MBAS2_STEP_NUM);

	//object 手自动切换
	IF (MBAS2.status.mode <> 0) AND (NOT MBAS2.auto_mode_edge) THEN
		MBAS2.auto_mode_edge := TRUE;
		MBAS2.manual_mode_edge := FALSE;

		MBALV0201.control.auto_operate := TRUE;
		STFLV0101.control.auto_operate := TRUE;
		STFLV0102.control.auto_operate := TRUE;
		STFP01.control.auto_operate := TRUE;
		MBAR03.control.auto_operate := TRUE;
		MBAXV0208.control.auto_operate := TRUE;
		MBATV0201B.control.auto_operate := TRUE;
		MBATV0201C.control.auto_operate := TRUE;
		MBATV0201F.control.auto_operate := TRUE;
		MBATV0201E.control.auto_operate := TRUE;
		MBAFQV0201.control.auto_operate := TRUE;
		MBAXV0207.control.auto_operate := TRUE;
		MBAXV1102.control.auto_operate := TRUE;
		MBAXV0209.control.auto_operate := TRUE;
	END_IF;

	IF (MBAS2.status.mode = 0) AND (NOT MBAS2.manual_mode_edge) THEN
		MBAS2.manual_mode_edge := TRUE;
		MBAS2.auto_mode_edge := FALSE;

		MBALV0201.control.manual_operate := TRUE;
		STFLV0101.control.manual_operate := TRUE;
		STFLV0102.control.manual_operate := TRUE;
		STFP01.control.manual_operate := TRUE;
		MBAR03.control.manual_operate := TRUE;
		MBAXV0208.control.manual_operate := TRUE;
		MBATV0201B.control.manual_operate := TRUE;
		MBATV0201C.control.manual_operate := TRUE;
		MBATV0201F.control.manual_operate := TRUE;
		MBATV0201E.control.manual_operate := TRUE;
		MBAFQV0201.control.manual_operate := TRUE;
		MBAXV0207.control.manual_operate := TRUE;
		MBAXV1102.control.manual_operate := TRUE;
		MBAXV0209.control.manual_operate := TRUE;
	END_IF;

	//错误信号停机
	MBAS2.input.error_signal := (MBALV0201.status.valve_status >= 2) OR (STFLV0101.status.valve_status >= 2) OR
	(STFLV0102.status.valve_status >= 2) OR (STFP01.status.motor_status >= 2) OR (MBAR03.status.motor_status >= 2) OR
	(MBAXV0208.status.valve_status >= 2) OR (MBATV0201B.status.valve_status >= 2) OR (MBATV0201C.status.valve_status >= 2) OR
	(MBATV0201F.status.valve_status >= 2) OR (MBATV0201E.status.valve_status >= 2) OR (MBAFQV0201.status.valve_status >= 2) OR
	(MBAXV0207.status.valve_status >= 2) OR (MBAXV1102.status.valve_status >= 2) OR (MBAXV0209.status.valve_status >= 2);

	IF MBAS2.status.run_state = 1 THEN
		//步骤执行动作
		CASE MBAS2.status.run_step OF
			0:
				IF NOT MBAS2_STEP[0].done THEN
					MBALV0201.control.auto_operate := TRUE;
					STFLV0101.control.auto_operate := TRUE;
					STFLV0102.control.auto_operate := TRUE;
					STFP01.control.auto_operate := TRUE;
					MBAR03.control.auto_operate := TRUE;
					MBAXV0208.control.auto_operate := TRUE;
					MBATV0201B.control.auto_operate := TRUE;
					MBATV0201C.control.auto_operate := TRUE;
					MBATV0201F.control.auto_operate := TRUE;
					MBATV0201E.control.auto_operate := TRUE;
					MBAFQV0201.control.auto_operate := TRUE;
					MBAXV0207.control.auto_operate := TRUE;
					MBAXV1102.control.auto_operate := TRUE;
					MBAXV0209.control.auto_operate := TRUE;
					MBAS2_STEP[0].done := TRUE;
				END_IF;
			1:
				CASE step2_1 OF
					0:
						IF NOT MBAS2_STEP[1].done THEN
							step2_1 := 1;
						END_IF;
					1:
						IF MBALIT0201.status.value <= MBAS2_PARA_L2 THEN
							step2_1 := 2;
						ELSE
							step2_1 := 6;
						END_IF;
					2:
						MBALV0201.input.auto_open_signal := TRUE;
						STFLV0101.input.auto_open_signal := FALSE;
						STFLV0102.input.auto_open_signal := FALSE;
						IF STFLV0101.input.close_feedback_state AND STFLV0102.input.close_feedback_state AND MBALV0201.input.open_feedback_state THEN
							step2_1 := 3;
						END_IF;
					3:
						LiquidAdd_3(level_value := MBALIT0201.status.value,
						sp_value := MBAS2_PARA_L1,
						sp_accumulation := MBAS2_PARA_AC1,
						sp_time := DINT_TO_TIME(MBAS2_PARA_T1 * 1000),
						flowmeter := STFFQIT0102,
						done := step2_1_3_done);
						STFP01.input.auto_run_signal := LiquidAdd_3.run;
						IF step2_1_3_done AND (NOT STFP01.input.run_feedback) AND (NOT STFP01.input.auto_run_signal) THEN
							step2_1 := 4;
						END_IF;
					4:
						IF STFFQIT0102.flowrate <= flowrate_threshold THEN
							step2_1 := 5;
						END_IF;
					5:
						MBALV0201.input.auto_open_signal := FALSE;
						IF MBALV0201.input.close_feedback_state THEN
							step2_1 := 6;
						END_IF;
					6:
						step2_1_3_done := FALSE;
						step2_1 := 0;
						MBAS2_STEP[1].done := TRUE;
				END_CASE;
			2:
				MBAR03.input.auto_run_signal := TRUE;
				IF MBAR03.input.run_feedback THEN
					MBAS2_STEP[2].done := TRUE;
				END_IF;
			3:
				LiquidRelease_4(sp_time := DINT_TO_TIME(MBAS2_PARA_T2 * 60 * 1000),
				level_value := MBALIT0201.status.value,
				set_point := MBAS2_PARA_L2,
				done := MBAS2_STEP[3].done);
				MBAXV0208.input.auto_open_signal := LiquidRelease_4.run;
			4:
				CASE step2_4 OF
					0:
						IF NOT MBAS2_STEP[4].done THEN
							step2_4 := 1;
						END_IF;
					1:
						HeatPot_0(ST1 := DINT_TO_TIME(MBAS2_PARA_T3 * 1000),
						ST2 := DINT_TO_TIME(MBAS2_PARA_T4 * 1000),
						V3 := MBATV0201B,
						V4 := MBATV0201C,
						V5 := MBATV0201F,
						V6 := MBATV0201E,
						done := step2_4_1_done);
						IF step2_4_1_done THEN
							step2_4 := 2;
						END_IF;
					2:
						IF MBATIT0201.status.value >= MBAS2_PARA_Temp1 THEN
							MBATV0201B.input.auto_open_signal := FALSE;
							step2_4 := 3;
						END_IF;
					3:
						IF MBATIT0201.status.value >= MBAS2_PARA_Temp2 THEN
							step2_4 := 4;
						END_IF;
					4:
						TON_1.PT := DINT_TO_TIME(MBAS2_PARA_T5 * 60 * 1000);
						TON_1.IN := TRUE;
						IF TON_1.Q THEN
							TON_1.IN := FALSE;
							step2_4 := 5;
						END_IF;
					5:
						MBATV0201C.input.auto_open_signal := FALSE;
						IF MBATV0201C.input.close_feedback_state THEN
							step2_4 := 0;
							step2_4_1_done := FALSE;
							MBAS2_STEP[4].done := TRUE;
						END_IF;
				END_CASE;
				TON_1();
			5:
				LiquidTransfer_1(sp_time := DINT_TO_TIME(MBAS2_PARA_T6 * 1000),
				sp_accumulation := MBAS2_PARA_AC2,
				done := MBAS2_STEP[5].done,
				flowmeter := MBAFQIT0503);
				MBAFQV0201.input.auto_open_signal := LiquidTransfer_1.run;
			6:
				//确认R13空闲
			7:
				MBAR03.input.auto_run_signal := FALSE;
				MBAXV1102.input.auto_open_signal := TRUE;
				IF (NOT MBAR03.input.run_feedback) AND MBAXV1102.input.open_feedback_state THEN
					MBAXV0207.input.auto_open_signal := TRUE;
					MBAS2_STEP[7].done := TRUE;
				END_IF;
			8:
				//确认转移完毕
			9:
				CASE step2_9 OF
					0:
						IF NOT MBAS2_STEP[9].done THEN
							step2_9 := 1;
						END_IF;
					1:
						LiquidTransfer_0(sp_time := DINT_TO_TIME(MBAS2_PARA_T7 * 1000),
						sp_accumulation := MBAS2_PARA_AC3,
						done := step2_9_1_done,
						flowmeter := MBAFQIT0503);
						MBAFQV0201.input.auto_open_signal := LiquidTransfer_0.run;
						IF step2_9_1_done AND MBAFQV0201.input.close_feedback_state AND (NOT MBAFQV0201.input.auto_open_signal) THEN
							step2_9 := 2;
						END_IF;
					2:
						TON_0.PT := DINT_TO_TIME(MBAS2_PARA_T8 * 1000);
						TON_0.IN := TRUE;
						IF TON_0.Q THEN
							TON_0.IN := FALSE;
							step2_9 := 3;
						END_IF;
					3:
						MBAXV0207.input.auto_open_signal := FALSE;
						MBAXV0209.input.auto_open_signal := FALSE;
						MBATV0201F.input.auto_open_signal := FALSE;
						IF MBAXV0207.input.close_feedback_state AND MBAXV0209.input.close_feedback_state AND MBATV0201F.input.close_feedback_state THEN
							step2_9 := 0;
							step2_9_1_done := FALSE;
							MBAS2_STEP[9].done := TRUE;
						END_IF;
				END_CASE;
				TON_0();
			10:
			//清理过滤器
		END_CASE;
	END_IF;

	//人工确认步骤可用
	IF (MBAS2.status.run_state) AND (NOT MBAS2_STEP[MBAS2.status.run_step].done AND ((MBAS2.status.run_step = 6) OR (MBAS2.status.run_step = 8) OR (MBAS2.status.run_step = 10))) THEN
		MBAS2.status.confirm_enable := TRUE;
	ELSE
		MBAS2.status.confirm_enable := FALSE;
	END_IF;
END_ACTION

(* ---- MBAS3_ACTION.st ---- *)
ACTION S3_ACT:
	//设定时间
	FOR i := 0 TO MBAS3_STEP_NUM DO
		IF MBAS3_ST[i] < T#5s THEN
			MBAS3_ST[i] := T#5s;
		END_IF;
		MBAS3_STEP[i].set_time := MBAS3_ST[i];
	END_FOR;

	//流程步骤
	ProcessHandleFC(MBAS3,MBAS3_STEP[0],MBAS3_STEP_NUM);

	//object 手自动切换
	IF (MBAS3.status.mode <> 0) AND (NOT MBAS3.auto_mode_edge) THEN
		MBAS3.auto_mode_edge := TRUE;
		MBAS3.manual_mode_edge := FALSE;

		MBAR04.control.auto_operate := TRUE;
		MBAXV0408.control.auto_operate := TRUE;
		MBAXV0409.control.auto_operate := TRUE;
		MBAFVT0401.control.auto_operate := TRUE;
		MBATV0401A.control.auto_operate := TRUE;
		MBATV0401B.control.auto_operate := TRUE;
		MBATV0401E.control.auto_operate := TRUE;
		MBATV0401F.control.auto_operate := TRUE;
		MBATV0401C.control.auto_operate := TRUE;
		MBATV0401D.control.auto_operate := TRUE;
		MBAXV0411.control.auto_operate := TRUE;
		MBAXV0415.control.auto_operate := TRUE;
	END_IF;

	IF (MBAS3.status.mode = 0) AND (NOT MBAS3.manual_mode_edge) THEN
		MBAS3.manual_mode_edge := TRUE;
		MBAS3.auto_mode_edge := FALSE;

		MBAR04.control.manual_operate := TRUE;
		MBAXV0408.control.manual_operate := TRUE;
		MBAXV0409.control.manual_operate := TRUE;
		MBAFVT0401.control.manual_operate := TRUE;
		MBATV0401A.control.manual_operate := TRUE;
		MBATV0401B.control.manual_operate := TRUE;
		MBATV0401E.control.manual_operate := TRUE;
		MBATV0401F.control.manual_operate := TRUE;
		MBATV0401C.control.manual_operate := TRUE;
		MBATV0401D.control.manual_operate := TRUE;
		MBAXV0411.control.manual_operate := TRUE;
		MBAXV0415.control.manual_operate := TRUE;
	END_IF;

	//错误信号停机
	MBAS3.input.error_signal := (MBAR04.status.motor_status >= 2) OR
	(MBAXV0408.status.valve_status >= 2) OR (MBAXV0409.status.valve_status >= 2) OR
	(MBATV0401A.status.valve_status >= 2) OR (MBATV0401B.status.valve_status >= 2) OR (MBAXV0415.status.valve_status >= 2) OR
	(MBATV0401E.status.valve_status >= 2) OR (MBATV0401F.status.valve_status >= 2) OR (MBATV0401C.status.valve_status >= 2) OR
	(MBATV0401D.status.valve_status >= 2) OR (MBAXV0411.status.valve_status >= 2);

	IF MBAS3.status.run_state = 1 THEN
		//步骤执行动作
		CASE MBAS3.status.run_step OF
			0:
				IF NOT MBAS3_STEP[0].done THEN
					MBAR04.control.auto_operate := TRUE;
					MBAXV0408.control.auto_operate := TRUE;
					MBAXV0409.control.auto_operate := TRUE;
					MBAFVT0401.control.auto_operate := TRUE;
					MBATV0401A.control.auto_operate := TRUE;
					MBATV0401B.control.auto_operate := TRUE;
					MBATV0401E.control.auto_operate := TRUE;
					MBATV0401F.control.auto_operate := TRUE;
					MBATV0401C.control.auto_operate := TRUE;
					MBATV0401D.control.auto_operate := TRUE;
					MBAXV0411.control.auto_operate := TRUE;
					MBAXV0415.control.auto_operate := TRUE;
					MBAS3_STEP[0].done := TRUE;
				END_IF;
			1:
				//确认皂化釜反应5批
			2:
				MBAR04.input.auto_run_signal := TRUE;
				MBAXV0409.input.auto_open_signal := TRUE;
				MBAXV0415.input.auto_open_signal := TRUE;
				MTBasicsPID_4.Enable := FALSE;
				MBAFVT0401.input.auto_degree_set := 0.0;
				IF MBAR04.input.run_feedback AND MBAXV0409.input.open_feedback_state AND MBAXV0415.input.open_feedback_state THEN
					MBAS3_STEP[2].done := TRUE;
				END_IF;
			3:
				CASE step3_3 OF
					0:
						IF NOT MBAS3_STEP[3].done THEN
							step3_3 := 1;
						END_IF;
					1:
						HeatPot_7(ST1 := DINT_TO_TIME(MBAS3_PARA_T1 * 1000),
						ST2 := DINT_TO_TIME(MBAS3_PARA_T2 * 1000),
						V3 := MBATV0401A,
						V4 := MBATV0401B,
						V5 := MBATV0401E,
						V6 := MBATV0401F,
						done := step3_3_1_done);
						IF step3_3_1_done THEN
							step3_3 := 2;
						END_IF;
					2:
						IF MBATIT0401.status.value >= MBAS3_PARA_Temp1 THEN
							step3_3 := 3;
						END_IF;
					3:
						MBATV0401A.input.auto_open_signal := FALSE;
						IF MBATV0401A.input.close_feedback_state THEN
							step3_3 := 0;
							step3_3_1_done := FALSE;
							MBAS3_STEP[3].done := TRUE;
						END_IF;
				END_CASE;
			4:
				CASE step3_4 OF
					0:
						last_value_MBATIT0402 := 0.0;
						IF NOT MBAS3_STEP[4].done THEN
							step3_4 := 1;
						END_IF;
//					1:
//						TON_2.PT := DINT_TO_TIME(MBAS3_PARA_T3 * 60 * 1000);
//						TON_2.IN := TRUE;
//						IF TON_2.Q THEN
//							TON_2.IN := FALSE;
//							IF ABS(MBATIT0402.status.value - last_value_MBATIT0402) <= MBAS3_PARA_Temp2 THEN
//								MTBasicsPID_4.Enable := TRUE;
////								MBAFVT0401.input.auto_degree_set := MBAS3_PARA_O2;
//								step3_4 := 2;
//							END_IF;
//							last_value_MBATIT0402 := MBATIT0402.status.value;
						//						END_IF;
					1:
						TON_2.PT := DINT_TO_TIME(MBAS3_PARA_T3 * 60 * 1000);
						IF MBATIT0402.status.value >= MBAS3_PARA_Temp2 THEN
							TON_2.IN := TRUE;
						END_IF;
						IF TON_2.Q THEN
							TON_2.IN := FALSE;
							MTBasicsPID_4.Enable := TRUE;
							step3_4 := 2;
						END_IF;
					2:
						IF MBATIT0401.status.value >= MBAS3_PARA_Temp3 THEN
							step3_4 := 3;
						END_IF;
					3:
						MBATV0401F.input.auto_open_signal := TRUE;
						IF MBATV0401F.input.open_feedback_state THEN
							step3_4 := 4;
						END_IF;
					4:
						MBATV0401B.input.auto_open_signal := FALSE;
						IF MBATV0401B.input.close_feedback_state THEN
							step3_4 := 5;
						END_IF;
					5:
						TON_2.PT := DINT_TO_TIME(MBAS3_PARA_T4 * 1000);
						TON_2.IN := TRUE;
						IF TON_2.Q THEN
							TON_2.IN := FALSE;
							step3_4 := 6;
						END_IF;
					6:
						MBATV0401E.input.auto_open_signal := FALSE;
						MBATV0401F.input.auto_open_signal := FALSE;
						IF MBATV0401E.input.close_feedback_state AND MBATV0401F.input.close_feedback_state THEN
							step3_4 := 0;
							MBAS3_STEP[4].done := TRUE;
						END_IF;
				END_CASE;
				TON_2();
				//手动控制出料阀
			5:
				CASE step3_5 OF
					0:
						IF NOT MBAS3_STEP[5].done THEN
							step3_5 := 1;
						END_IF;
					1:
						MBATV0401C.input.auto_open_signal := TRUE;
						IF MBATV0401C.input.open_feedback_state THEN
							step3_5 := 2;
						END_IF;
					2:
						MBATV0401D.input.auto_open_signal := TRUE;
						IF MBATV0401D.input.open_feedback_state THEN
							step3_5 := 3;
						END_IF;
					3:
						IF MBATIT0401.status.value <= MBAS3_PARA_Temp4 THEN
							step3_5 := 4;
						END_IF;
					4:
						MBATV0401D.input.auto_open_signal := FALSE;
						IF MBATV0401D.input.close_feedback_state THEN
							step3_5 := 5;
						END_IF;
					5:
						MBATV0401C.input.auto_open_signal := FALSE;
						IF MBATV0401C.input.close_feedback_state THEN
							step3_5 := 6;
						END_IF;
					6:
						MBAR04.input.auto_run_signal := FALSE;
						IF NOT MBAR04.input.run_feedback THEN
							step3_5 := 7;
						END_IF;
					7:
						MTBasicsPID_4.Enable := FALSE;
						MBAFVT0401.input.auto_degree_set := 0.0;
						MBAXV0409.input.auto_open_signal := FALSE;
						IF MBAXV0409.input.close_feedback_state THEN
							step3_5 := 0;
							MBAS3_STEP[5].done := TRUE;
						END_IF;
				END_CASE;
			6:
				CASE step3_9 OF
					0:
						IF NOT MBAS3_STEP[6].done THEN
							step3_9 := 1;
						END_IF;
					1:
						MBAXV0411.input.auto_open_signal := TRUE;
						step3_9 := 2;
					2:
						IF MBALIT0401.status.value <= 0.0 THEN
							step3_9 := 3;
						END_IF;
					3:
						TON_4.PT := DINT_TO_TIME(MBAS3_PARA_T5 * 60 * 1000);
						TON_4.IN := TRUE;
						IF TON_4.Q THEN
							TON_4.IN := FALSE;
							step3_9 := 4;
						END_IF;
					4:
						MBAXV0411.input.auto_open_signal := FALSE;
						IF MBAXV0411.input.close_feedback_state THEN
							step3_9 := 0;
							MBAS3_STEP[6].done := TRUE;
						END_IF;
				END_CASE;
				TON_4();
		END_CASE;
	END_IF;

	//FVT0401 pid调节
	R_TRIG_4(CLK := MBAFVT0401.status.auto_mode);
	IF R_TRIG_4.Q THEN
		MTBasicsPID_4.Enable := TRUE;
	END_IF;
	F_TRIG_4(CLK := MBAFVT0401.status.auto_mode);
	IF F_TRIG_4.Q THEN
		MTBasicsPID_4.Enable := FALSE;
	END_IF;
	//MTBasicsPID_4.Enable := TRUE;
	MTBasicsPID_4.PIDParameters.Gain := MBAPidFVT0401Para.gain;
	MTBasicsPID_4.PIDParameters.IntegrationTime := MBAPidFVT0401Para.integration_time;
	MTBasicsPID_4.PIDParameters.DerivativeTime := MBAPidFVT0401Para.derivative_time;
	MTBasicsPID_4.MinOut := 0.0;
	MTBasicsPID_4.MaxOut := 100.0;
	MTBasicsPID_4.SetValue := MBAPidFVT0401Para.set_value;
	MTBasicsPID_4.ActValue := MBAFIT0401.flowrate;
	MTBasicsPID_4.Update := MBAPidFVT0401.update;
	MTBasicsPID_4();
	MBAPidFVT0401.out := MTBasicsPID_4.Out;
	IF MTBasicsPID_4.Active THEN
		MBAFVT0401.input.auto_degree_set := MTBasicsPID_4.Out + MBAPidFVT0401Para.min_out;
		//	ELSE
		//		MBAFVT0401.input.auto_degree_set := 0.0;
	END_IF;
	IF MTBasicsPID_4.UpdateDone THEN
		MBAPidFVT0401.update := FALSE;
	END_IF;

	//人工确认步骤可用
	IF (MBAS3.status.run_state) AND (NOT MBAS3_STEP[MBAS3.status.run_step].done AND ((MBAS3.status.run_step = 1))) THEN
		MBAS3.status.confirm_enable := TRUE;
	ELSE
		MBAS3.status.confirm_enable := FALSE;
	END_IF;
END_ACTION

(* ---- MBAS4_ACTION.st ---- *)
ACTION S4_ACT:
	//设定时间
	FOR i := 0 TO MBAS4_STEP_NUM DO
		IF MBAS4_ST[i] < T#5s THEN
			MBAS4_ST[i] := T#5s;
		END_IF;
		MBAS4_STEP[i].set_time := MBAS4_ST[i];
	END_FOR;

	//流程步骤
	ProcessHandleFC(MBAS4,MBAS4_STEP[0],MBAS4_STEP_NUM);

	//object 手自动切换
	IF (MBAS4.status.mode <> 0) AND (NOT MBAS4.auto_mode_edge) THEN
		MBAS4.auto_mode_edge := TRUE;
		MBAS4.manual_mode_edge := FALSE;
		//
		STFLV0301.control.auto_operate := TRUE;
		STFLV0302.control.auto_operate := TRUE;
		MBALV0301.control.auto_operate := TRUE;
		STFP03.control.auto_operate := TRUE;
		MBAFQV0301.control.auto_operate := TRUE;
		MBAXV0306.control.auto_operate := TRUE;
		MBAR07.control.auto_operate := TRUE;
		MBATV0301.control.auto_operate := TRUE;
		MBAAV0301.control.auto_operate := TRUE;
		MBAXV0627.control.auto_operate := TRUE;
		MBAXV0629.control.auto_operate := TRUE;
		MBAXV0630.control.auto_operate := TRUE;
	END_IF;

	IF (MBAS4.status.mode = 0) AND (NOT MBAS4.manual_mode_edge) THEN
		MBAS4.manual_mode_edge := TRUE;
		MBAS4.auto_mode_edge := FALSE;

		STFLV0301.control.manual_operate := TRUE;
		STFLV0302.control.manual_operate := TRUE;
		MBALV0301.control.manual_operate := TRUE;
		STFP03.control.manual_operate := TRUE;
		MBAFQV0301.control.manual_operate := TRUE;
		MBAXV0306.control.manual_operate := TRUE;
		MBAR07.control.manual_operate := TRUE;
		MBATV0301.control.manual_operate := TRUE;
		MBAAV0301.control.manual_operate := TRUE;
		MBAXV0627.control.manual_operate := TRUE;
		MBAXV0629.control.manual_operate := TRUE;
		MBAXV0630.control.manual_operate := TRUE;
	END_IF;

	//错误信号停机
	MBAS4.input.error_signal := (STFLV0301.status.valve_status >= 2) OR (STFLV0302.status.valve_status >= 2) OR
	(MBALV0301.status.valve_status >= 2) OR (STFP03.status.motor_status >= 2) OR (MBAFQV0301.status.valve_status >= 2) OR
	(MBAXV0306.status.valve_status >= 2) OR (MBAR07.status.motor_status >= 2) OR (MBATV0301.status.valve_status >= 2) OR
	(MBAAV0301.status.valve_status >= 2) OR (MBAXV0627.status.valve_status >= 2) OR
	(MBAXV0629.status.valve_status >= 2) OR (MBAXV0630.status.valve_status >= 2);

	IF MBAS4.status.run_state = 1 THEN
		//步骤执行动作
		CASE MBAS4.status.run_step OF
			0:
				IF NOT MBAS4_STEP[0].done THEN
					STFLV0301.control.auto_operate := TRUE;
					STFLV0302.control.auto_operate := TRUE;
					MBALV0301.control.auto_operate := TRUE;
					STFP03.control.auto_operate := TRUE;
					MBAFQV0301.control.auto_operate := TRUE;
					MBAXV0306.control.auto_operate := TRUE;
					MBAR07.control.auto_operate := TRUE;
					MBATV0301.control.auto_operate := TRUE;
					MBAAV0301.control.auto_operate := TRUE;
					MBAXV0627.control.auto_operate := TRUE;
					MBAXV0629.control.auto_operate := TRUE;
					MBAXV0630.control.auto_operate := TRUE;
					MBAS4_STEP[0].done := TRUE;
				END_IF;
			1:
				CASE step4_1 OF
					0:
						IF NOT MBAS4_STEP[1].done THEN
							step4_1 := 1;
						END_IF;
					1:
						STFLV0301.input.auto_open_signal := TRUE;
						STFLV0302.input.auto_open_signal := FALSE;
						MBALV0301.input.auto_open_signal := TRUE;
						IF MBALV0301.input.open_feedback_state AND STFLV0301.input.open_feedback_state AND STFLV0302.input.close_feedback_state THEN
							step4_1 := 2;
						END_IF;
					2:
						LiquidAdd_7(level_value := MBALIT0301.status.value,
						sp_value := MBAS4_PARA_L4,
						sp_accumulation := MBAS4_PARA_AC1,
						sp_time := DINT_TO_TIME(MBAS4_PARA_T1 * 1000),
						flowmeter := STFFQIT0302,
						done := step4_1_2_done);
						STFP03.input.auto_run_signal := LiquidAdd_7.run;
						IF step4_1_2_done AND (NOT STFP03.input.run_feedback) AND (NOT STFP03.input.auto_run_signal) THEN
							step4_1 := 3;
						END_IF;
					3:
						IF STFFQIT0302.flowrate <= flowrate_threshold THEN
							step4_1 := 4;
						END_IF;
					4:
						MBALV0301.input.auto_open_signal := FALSE;
						IF MBALV0301.input.close_feedback_state THEN
							step4_1 := 0;
							step4_1_2_done := FALSE;
							MBAS4_STEP[1].done := TRUE;
						END_IF;
				END_CASE;
			2:
				//加水
				LiquidTransfer_2(sp_time := DINT_TO_TIME(MBAS4_PARA_T5 * 1000),
				sp_accumulation := MBAS4_PARA_AC2,
				done := MBAS4_STEP[2].done,
				flowmeter := MBAFQIT0503);
				MBAFQV0301.input.auto_open_signal := LiquidTransfer_2.run;
			3:
				//滴加
				CASE step4_3 OF
					0:
						IF NOT MBAS4_STEP[3].done THEN
							step4_3 := 1;
						END_IF;
					1:
						MBAXV0306.input.auto_open_signal := TRUE;
						MBAR07.input.auto_run_signal := TRUE;
						IF MBAXV0306.input.open_feedback_state AND MBAR07.input.run_feedback THEN
							step4_3 := 2;
						END_IF;
					2:
						IF MBALIT0301.status.value > 0.0 THEN
							IF MBATIT0301.status.value <= MBAS4_PARA_Temp1 THEN
								MBATV0301.input.auto_open_signal := TRUE;
							END_IF;
							IF MBATIT0301.status.value >= MBAS4_PARA_Temp2 THEN
								MBATV0301.input.auto_open_signal := FALSE;
							END_IF;
						ELSE
							step4_3 := 3;
						END_IF;
					3:
						TON_16.PT := DINT_TO_TIME(MBAS4_PARA_T6 * 1000);
						TON_16.IN := TRUE;
						IF TON_16.Q THEN
							TON_16.IN := FALSE;
							step4_3 := 4;
						END_IF;
					4:
						MBATV0301.input.auto_open_signal := FALSE;
						MBAXV0306.input.auto_open_signal := FALSE;
						MBAR07.input.auto_run_signal := FALSE;
						IF MBATV0301.input.close_feedback_state AND MBAXV0306.input.close_feedback_state AND (NOT MBAR07.input.run_feedback) THEN
							step4_3 := 0;
							MBAS4_STEP[3].done := TRUE;
						END_IF;
				END_CASE;
				TON_16();
		END_CASE;
	END_IF;

	//人工确认步骤可用
	//	IF (MBAS4.status.run_state) AND (NOT MBAS4_STEP[MBAS4.status.run_step].done AND ((MBAS4.status.run_step = 1) OR (MBAS4.status.run_step = 2) OR (MBAS4.status.run_step = 4))) THEN
	//		MBAS4.status.confirm_enable := TRUE;
	//	ELSE
	//		MBAS4.status.confirm_enable := FALSE;
	//	END_IF;
END_ACTION

(* ---- MBAS5_ACTION.st ---- *)
ACTION S5_ACT:
	//设定时间
	FOR i := 0 TO MBAS5_STEP_NUM DO
		IF MBAS5_ST[i] < T#5s THEN
			MBAS5_ST[i] := T#5s;
		END_IF;
		MBAS5_STEP[i].set_time := MBAS5_ST[i];
	END_FOR;

	//流程步骤
	ProcessHandleFC(MBAS5,MBAS5_STEP[0],MBAS5_STEP_NUM);

	//object 手自动切换
	IF (MBAS5.status.mode <> 0) AND (NOT MBAS5.auto_mode_edge) THEN
		MBAS5.auto_mode_edge := TRUE;
		MBAS5.manual_mode_edge := FALSE;

		MBAXV0308.control.auto_operate := TRUE;
		MBAXV0301.control.auto_operate := TRUE;
		MBAR13.control.auto_operate := TRUE;
		MBAPHV1101.control.auto_operate := TRUE;
		MBATV1101.control.auto_operate := TRUE;
	END_IF;

	IF (MBAS5.status.mode = 0) AND (NOT MBAS5.manual_mode_edge) THEN
		MBAS5.manual_mode_edge := TRUE;
		MBAS5.auto_mode_edge := FALSE;

		MBAXV0308.control.manual_operate := TRUE;
		MBAXV0301.control.manual_operate := TRUE;
		MBAR13.control.manual_operate := TRUE;
		MBAPHV1101.control.manual_operate := TRUE;
		MBATV1101.control.manual_operate := TRUE;
	END_IF;

	//错误信号停机
	MBAS5.input.error_signal := (MBAXV0308.status.valve_status >= 2) OR (MBAXV0301.status.valve_status >= 2) OR
	(MBAR13.status.motor_status >= 2) OR (MBAPHV1101.status.valve_status >= 2) OR (MBATV1101.status.valve_status >= 2);

	IF MBAS5.status.run_state = 1 THEN
		//步骤执行动作
		CASE MBAS5.status.run_step OF
			0:
				IF NOT MBAS5_STEP[0].done THEN
					MBAXV0308.control.auto_operate := TRUE;
					MBAXV0301.control.auto_operate := TRUE;
					MBAR13.control.auto_operate := TRUE;
					MBAPHV1101.control.auto_operate := TRUE;
					MBATV1101.control.auto_operate := TRUE;
					MBAS5_STEP[0].done := TRUE;
				END_IF;
			1:
				//V30进料
				IF MBALIT1101.status.value >= MBAS5_PARA_L1 THEN
					MBAXV0308.input.auto_open_signal := FALSE;
					MBAXV0301.input.auto_open_signal := FALSE;
					MBAS5_STEP[1].done := TRUE;
				ELSE
					MBAXV0308.input.auto_open_signal := TRUE;
					MBAXV0301.input.auto_open_signal := TRUE;
				END_IF;
			2:
				//酸化
				CASE step5_2 OF
					0:
						IF NOT MBAS5_STEP[2].done THEN
							step5_2 := 1;
						END_IF;
					1:
						MBAR13.input.auto_run_signal := TRUE;
						IF MBAR13.input.run_feedback THEN
							step5_2 := 2;
						END_IF;
					2:
						TON_17.PT := DINT_TO_TIME(MBAS5_PARA_T3 * 1000);
						TON_17.IN := TRUE;
						IF TON_17.Q THEN
							TON_17.IN := FALSE;
							step5_2 := 3;
						END_IF;
					3:
						MBAPHV1101.input.auto_open_signal := TRUE;
						IF MBAPHV1101.input.open_feedback_state THEN
							temp_monitor_0302 := TRUE;
							step5_2 := 4;
						END_IF;
					4:
						TON_17.PT := DINT_TO_TIME(MBAS5_PARA_T4 * 60 * 1000);
						TON_17.IN := TRUE;
						IF TON_17.Q THEN
							TON_17.IN := FALSE;
							step5_2 := 5;
						END_IF;
					5:
						MBAPHV1101.input.auto_open_signal := FALSE;
						temp_monitor_0302 := FALSE;
						IF MBAPHV1101.input.close_feedback_state THEN
							MBATV1101.input.auto_open_signal := FALSE;
							IF MBATV1101.input.close_feedback_state THEN
								step5_2 := 6;
							END_IF;
						END_IF;
					6:
						TON_17.PT := DINT_TO_TIME(MBAS5_PARA_T5 * 60 * 1000);
						TON_17.IN := TRUE;
						IF TON_17.Q THEN
							TON_17.IN := FALSE;
							step5_2 := 0;
							MBAS5_STEP[2].done := TRUE;
						END_IF;
				END_CASE;
				TON_17();
			3:
				//离心
		END_CASE;
	END_IF;

	//V06滴加温控
	IF temp_monitor_0302 THEN
		IF MBATIT1101.status.value >= MBAS5_PARA_Temp1 THEN
			MBATV1101.input.auto_open_signal := TRUE;
		END_IF;
		IF MBATIT1101.status.value <= MBAS5_PARA_Temp2 THEN
			MBATV1101.input.auto_open_signal := FALSE;
		END_IF;
	END_IF;

	//人工确认步骤可用
	IF (MBAS5.status.run_state) AND (NOT MBAS5_STEP[MBAS5.status.run_step].done AND ((MBAS5.status.run_step = 3))) THEN
		MBAS5.status.confirm_enable := TRUE;
	ELSE
		MBAS5.status.confirm_enable := FALSE;
	END_IF;

END_ACTION

(* ---- MBAS6_ACTION.st ---- *)
ACTION S6_ACT:
	//设定时间
	FOR i := 0 TO MBAS6_STEP_NUM DO
		IF MBAS6_ST[i] < T#5s THEN
			MBAS6_ST[i] := T#5s;
		END_IF;
		MBAS6_STEP[i].set_time := MBAS6_ST[i];
	END_FOR;

	//流程步骤
	ProcessHandleFC(MBAS6,MBAS6_STEP[0],MBAS6_STEP_NUM);

	//object 手自动切换
	IF (MBAS6.status.mode <> 0) AND (NOT MBAS6.auto_mode_edge) THEN
		MBAS6.auto_mode_edge := TRUE;
		MBAS6.manual_mode_edge := FALSE;

		MBAXV0510.control.auto_operate := TRUE;
		MBAXV0526.control.auto_operate := TRUE;
		MBAXV0507.control.auto_operate := TRUE;
		MBAR02.control.auto_operate := TRUE;
		MBAXV0305.control.auto_operate := TRUE;
		MBAAV0301.control.auto_operate := TRUE;
		MBAXV0517.control.auto_operate := TRUE;
		MBATV0501C.control.auto_operate := TRUE;
		MBATV0501B.control.auto_operate := TRUE;
		MBATV0501E.control.auto_operate := TRUE;
		MBATV0501F.control.auto_operate := TRUE;
		MBAXV0515.control.auto_operate := TRUE;
		MBAXV0518.control.auto_operate := TRUE;
		MBAXV0512.control.auto_operate := TRUE;
		MBAXV0514.control.auto_operate := TRUE;
		MBAXV0524.control.auto_operate := TRUE;
	END_IF;

	IF (MBAS6.status.mode = 0) AND (NOT MBAS6.manual_mode_edge) THEN
		MBAS6.manual_mode_edge := TRUE;
		MBAS6.auto_mode_edge := FALSE;

		MBAXV0510.control.manual_operate := TRUE;
		MBAXV0526.control.manual_operate := TRUE;
		MBAXV0507.control.manual_operate := TRUE;
		MBAR02.control.manual_operate := TRUE;
		MBAXV0305.control.manual_operate := TRUE;
		MBAAV0301.control.manual_operate := TRUE;
		MBAXV0517.control.manual_operate := TRUE;
		MBATV0501C.control.manual_operate := TRUE;
		MBATV0501B.control.manual_operate := TRUE;
		MBATV0501E.control.manual_operate := TRUE;
		MBATV0501F.control.manual_operate := TRUE;
		MBAXV0515.control.manual_operate := TRUE;
		MBAXV0518.control.manual_operate := TRUE;
		MBAXV0512.control.manual_operate := TRUE;
		MBAXV0514.control.manual_operate := TRUE;
		MBAXV0524.control.manual_operate := TRUE;
	END_IF;

	//错误信号停机
	MBAS6.input.error_signal := (MBAXV0510.status.valve_status >= 2) OR (MBAXV0526.status.valve_status >= 2) OR
	(MBAR02.status.motor_status >= 2) OR (MBAXV0507.status.valve_status >= 2) OR (MBAXV0305.status.valve_status >= 2) OR
	(MBAAV0301.status.valve_status >= 2) OR (MBAXV0517.status.valve_status >= 2) OR (MBATV0501C.status.valve_status >= 2) OR
	(MBATV0501B.status.valve_status >= 2) OR (MBATV0501E.status.valve_status >= 2) OR (MBATV0501F.status.valve_status >= 2) OR
	(MBAXV0515.status.valve_status >= 2) OR (MBAXV0518.status.valve_status >= 2) OR (MBAXV0512.status.valve_status >= 2) OR
	(MBAXV0514.status.valve_status >= 2) OR (MBAXV0524.status.valve_status >= 2);

	IF MBAS6.status.run_state = 1 THEN
		//步骤执行动作
		CASE MBAS6.status.run_step OF
			0:
				MBAXV0510.control.auto_operate := TRUE;
				MBAXV0526.control.auto_operate := TRUE;
				MBAXV0507.control.auto_operate := TRUE;
				MBAR02.control.auto_operate := TRUE;
				MBAXV0305.control.auto_operate := TRUE;
				MBAAV0301.control.auto_operate := TRUE;
				MBAXV0517.control.auto_operate := TRUE;
				MBATV0501C.control.auto_operate := TRUE;
				MBATV0501B.control.auto_operate := TRUE;
				MBATV0501E.control.auto_operate := TRUE;
				MBATV0501F.control.auto_operate := TRUE;
				MBAXV0515.control.auto_operate := TRUE;
				MBAXV0518.control.auto_operate := TRUE;
				MBAXV0512.control.auto_operate := TRUE;
				MBAXV0514.control.auto_operate := TRUE;
				MBAXV0524.control.auto_operate := TRUE;
				//				is_liquid_R06 := 0;
				is_press_ok_R06 := FALSE;
				//				popup_is_liquid_R06 := FALSE;
				step9_temp_enable := FALSE;
				MBAS6_STEP[0].done := TRUE;
			1:
				//R02进料
			2:
				//试漏
			3:
				//进料
				CASE step6_3 OF
					0:
						IF NOT MBAS6_STEP[3].done THEN
							step6_3 := 1;
						END_IF;
					1:
						MBAR02.input.auto_run_signal := TRUE;
						TON_9.PT := DINT_TO_TIME(MBAS6_PARA_T2 * 60 * 1000);
						TON_9.IN := TRUE;
						IF TON_9.Q THEN
							TON_9.IN := FALSE;
							step6_3 := 2;
						END_IF;
					2:
						MBAXV0305.input.auto_open_signal := TRUE;
						IF MBAXV0305.input.open_feedback_state THEN
							step6_3 := 3;
						END_IF;
					3:
						IF MBAPIT0501.status.value <= MBAS6_PARA_P3 THEN
							MBAXV0510.input.auto_open_signal := TRUE;
							step6_3 := 4;
						END_IF;
					4:
						TON_9.PT := DINT_TO_TIME(MBAS6_PARA_T3 * 60 * 1000);
						TON_9.IN := TRUE;
						IF TON_9.Q THEN
							TON_9.IN := FALSE;
							MBAS6_STEP[3].done := TRUE;
							step6_3 := 0;
						END_IF;
				END_CASE;
				TON_9();
			4:
				//确认R02转移完毕
			5:
				MBAR02.input.auto_run_signal := FALSE;
				MBAS6_STEP[5].done := TRUE;
			6:
				//清洗管线
				TON_21.PT := DINT_TO_TIME(MBAS6_PARA_T4 * 60 * 1000);
				IF NOT MBAS6_STEP[6].done THEN
					MBAAV0301.input.auto_open_signal := TRUE;
					IF MBAAV0301.input.open_feedback_state THEN
						TON_21.IN := TRUE;
					END_IF;
				END_IF;
				IF TON_21.Q THEN
					TON_21.IN := FALSE;
					MBAXV0305.input.auto_open_signal := FALSE;
					MBAAV0301.input.auto_open_signal := FALSE;
					MBAS6_STEP[6].done := TRUE;
				END_IF;
				TON_21();
				//========================溶解==========================
			7:
				//准备 人工打开MBAR06搅拌
				MBAXV0517.input.auto_open_signal := TRUE;
			8:
				HeatPot_2(ST1 := DINT_TO_TIME(MBAS6_PARA_T5 * 1000),
				ST2 := DINT_TO_TIME(MBAS6_PARA_T6 * 1000),
				V3 := MBATV0501C,
				V4 := MBATV0501B,
				V5 := MBATV0501E,
				V6 := MBATV0501F,
				done := MBAS6_STEP[8].done);
			9:
				IF MBATIT0501.status.value >= MBAS6_PARA_Temp1 THEN
					MBATV0501C.input.auto_open_signal := FALSE;
					MBAXV0510.input.auto_open_signal := FALSE;
					step9_temp_enable := TRUE;
					IF MBATV0501C.input.close_feedback_state AND MBAXV0510.input.close_feedback_state THEN
						MBAS6_STEP[9].done := TRUE;
					END_IF;
				END_IF;
			10:
				//现场观察溶解清透 R08空闲
			11:
				step9_temp_enable := FALSE;
				MBATV0501B.input.auto_open_signal := FALSE;
				MBATV0501E.input.auto_open_signal := FALSE;
				MBATV0501F.input.auto_open_signal := TRUE;
				IF MBATV0501B.input.close_feedback_state AND MBATV0501E.input.close_feedback_state AND MBATV0501F.input.open_feedback_state THEN
					MBAS6_STEP[11].done := TRUE;
				END_IF;
			12:
				MBAXV0515.input.auto_open_signal := TRUE;
				MBAXV0518.input.auto_open_signal := TRUE;
				MBAXV0512.input.auto_open_signal := TRUE;
				MBAXV0524.input.auto_open_signal := TRUE;
				IF MBAXV0515.input.open_feedback_state AND MBAXV0518.input.open_feedback_state AND MBAXV0512.input.open_feedback_state AND MBAXV0524.input.open_feedback_state THEN
					MBAS6_STEP[12].done := TRUE;
				END_IF;
			13:
				CASE step6_13 OF
					0:
						IF NOT MBAS6_STEP[13].done THEN
							step6_13 := 1;
						END_IF;
					1:
						MBAXV0526.input.auto_open_signal := TRUE;
						step6_13 := 2;
					2:
						IF MBAPIT0501.status.value <= MBAS6_PARA_P6 THEN
							MBAXV0526.input.auto_open_signal := FALSE;
							MBAXV0514.input.auto_open_signal := TRUE;
							step6_13 := 3;
						END_IF;
					3:
						IF MBAXV0514.input.open_feedback_state THEN
							step6_13 := 0;
							MBAS6_STEP[13].done := TRUE;
						END_IF;
				END_CASE;
			14:
				IF MBATIT0501.status.value >= MBAS6_PARA_Temp5 THEN
					MBATV0501F.input.auto_open_signal := TRUE;
					IF MBATV0501F.input.open_feedback_state THEN
						MBATV0501B.input.auto_open_signal := FALSE;
						IF MBATV0501B.input.close_feedback_state THEN
							MBATV0501E.input.auto_open_signal := FALSE;
						END_IF;
					END_IF;
				ELSIF MBATIT0501.status.value <= MBAS6_PARA_Temp4 THEN
					MBATV0501E.input.auto_open_signal := TRUE;
					MBATV0501F.input.auto_open_signal := FALSE;
					IF MBATV0501E.input.open_feedback_state THEN
						MBATV0501B.input.auto_open_signal := TRUE;
					END_IF;
				END_IF;
				IF MBAPIT0501.status.value >= MBAS6_PARA_P7 THEN
					MBAXV0526.input.auto_open_signal := TRUE;
				ELSIF MBAPIT0501.status.value <= MBAS6_PARA_P8 THEN
					MBAXV0526.input.auto_open_signal := FALSE;
				END_IF;
				//观察R08进料管
			15:
				MBATV0501B.input.auto_open_signal := FALSE;
				IF MBATV0501B.input.close_feedback_state THEN
					MBATV0501E.input.auto_open_signal := FALSE;
				END_IF;
				MBATV0501F.input.auto_open_signal := TRUE;
				MBAXV0514.input.auto_open_signal := FALSE;
				MBAXV0512.input.auto_open_signal := FALSE;
				MBAXV0526.input.auto_open_signal := FALSE;
				//手动停R06
			16:
			//清理
		END_CASE;
	END_IF;

	//step9 温控
	IF step9_temp_enable THEN
		IF MBATIT0501.status.value >= MBAS6_PARA_Temp2 OR MBAPIT0501.status.value >= MBAS6_PARA_P4 THEN
			MBATV0501B.input.auto_open_signal := FALSE;
		ELSIF MBATIT0501.status.value <= MBAS6_PARA_Temp3 OR MBAPIT0501.status.value <= MBAS6_PARA_P5 THEN
			MBATV0501B.input.auto_open_signal := TRUE;
		END_IF;
	END_IF;

	//R06试漏
	IF press_test_R06 THEN
		CASE step6_2 OF
			0:
				MBAXV0510.control.auto_operate := TRUE;
				MBAXV0526.control.auto_operate := TRUE;
				MBAXV0507.control.auto_operate := TRUE;
				is_press_ok_R06 := FALSE;
				step6_2 := 1;
			1:
				MBAXV0510.input.auto_open_signal := FALSE;
				MBAXV0526.input.auto_open_signal := FALSE;
				IF MBAXV0510.input.close_feedback_state AND MBAXV0526.input.close_feedback_state THEN
					step6_2 := 2;
				END_IF;
			2:
				MBAXV0507.input.auto_open_signal := TRUE;
				step6_2 := 3;
			3:
				IF MBAPIT0501.status.value >= MBAS6_PARA_P1 THEN
					MBAXV0507.input.auto_open_signal := FALSE;
					step6_2 := 4;
				END_IF;
			4:
				TON_3.PT := DINT_TO_TIME(MBAS6_PARA_T1 * 60 * 1000);
				TON_3.IN := TRUE;
				IF TON_3.Q THEN
					TON_3.IN := FALSE;
					step6_2 := 5;
				END_IF;
			5:
				IF MBAS6_PARA_P1 - MBAPIT0501.status.value <= MBAS6_PARA_P2 THEN
					is_press_ok_R06 := TRUE;
				ELSE
					is_press_ok_R06 := FALSE;
				END_IF;
				step6_2 := 6;
			6:
				press_test_R06 := FALSE;
				step6_2 := 0;
		END_CASE;
		TON_3();
	END_IF;

	//人工确认步骤可用
	IF (MBAS6.status.run_state) AND (NOT MBAS6_STEP[MBAS6.status.run_step].done AND ((MBAS6.status.run_step = 1) OR (MBAS6.status.run_step = 2) OR (MBAS6.status.run_step = 4) OR (MBAS6.status.run_step = 7) OR (MBAS6.status.run_step = 10) OR
		(MBAS6.status.run_step = 14) OR (MBAS6.status.run_step = 15) OR (MBAS6.status.run_step = 16))) THEN
		MBAS6.status.confirm_enable := TRUE;
	ELSE
		MBAS6.status.confirm_enable := FALSE;
	END_IF;
END_ACTION

(* ---- MBAS7_ACTION.st ---- *)
ACTION S7_ACT:
	//设定时间
	FOR i := 0 TO MBAS7_STEP_NUM DO
		IF MBAS7_ST[i] < T#5s THEN
			MBAS7_ST[i] := T#5s;
		END_IF;
		MBAS7_STEP[i].set_time := MBAS7_ST[i];
	END_FOR;

	//流程步骤
	ProcessHandleFC(MBAS7,MBAS7_STEP[0],MBAS7_STEP_NUM);

	//object 手自动切换
	IF (MBAS7.status.mode <> 0) AND (NOT MBAS7.auto_mode_edge) THEN
		MBAS7.auto_mode_edge := TRUE;
		MBAS7.manual_mode_edge := FALSE;

		MBAXV0515.control.auto_operate := TRUE;
		MBAXV0518.control.auto_operate := TRUE;
		MBAXV0512.control.auto_operate := TRUE;
		MBAXV0524.control.auto_operate := TRUE;
		MBAXV0526.control.auto_operate := TRUE;
		MBAXV0514.control.auto_operate := TRUE;
		MBATV0501C.control.auto_operate := TRUE;
		MBATV0501E.control.auto_operate := TRUE;
		MBATV0501F.control.auto_operate := TRUE;
		MBAXV0519.control.auto_operate := TRUE;
		MBAXV0517.control.auto_operate := TRUE;
		MBATVT0510.control.auto_operate := TRUE;
	END_IF;

	IF (MBAS7.status.mode = 0) AND (NOT MBAS7.manual_mode_edge) THEN
		MBAS7.manual_mode_edge := TRUE;
		MBAS7.auto_mode_edge := FALSE;

		MBAXV0515.control.manual_operate := TRUE;
		MBAXV0518.control.manual_operate := TRUE;
		MBAXV0512.control.manual_operate := TRUE;
		MBAXV0524.control.manual_operate := TRUE;
		MBAXV0526.control.manual_operate := TRUE;
		MBAXV0514.control.manual_operate := TRUE;
		MBATV0501C.control.manual_operate := TRUE;
		MBATV0501E.control.manual_operate := TRUE;
		MBATV0501F.control.manual_operate := TRUE;
		MBAXV0519.control.manual_operate := TRUE;
		MBAXV0517.control.manual_operate := TRUE;
		MBATVT0510.control.manual_operate := TRUE;
	END_IF;

	//错误信号停机
	MBAS7.input.error_signal := (MBAXV0515.status.valve_status >= 2) OR (MBAXV0518.status.valve_status >= 2) OR
	(MBAXV0512.status.valve_status >= 2) OR (MBAXV0524.status.valve_status >= 2) OR (MBAXV0526.status.valve_status >= 2) OR
	(MBAXV0514.status.valve_status >= 2) OR (MBATV0501C.status.valve_status >= 2) OR (MBATV0501E.status.valve_status >= 2) OR
	(MBATV0501F.status.valve_status >= 2) OR (MBAXV0519.status.valve_status >= 2) OR (MBAXV0517.status.valve_status >= 2);

	IF MBAS7.status.run_state = 1 THEN
		//步骤执行动作
		CASE MBAS7.status.run_step OF
			0:
				IF NOT MBAS7_STEP[0].done THEN
					MBAXV0515.control.auto_operate := TRUE;
					MBAXV0518.control.auto_operate := TRUE;
					MBAXV0512.control.auto_operate := TRUE;
					MBAXV0524.control.auto_operate := TRUE;
					MBAXV0526.control.auto_operate := TRUE;
					MBAXV0514.control.auto_operate := TRUE;
					MBATV0501C.control.auto_operate := TRUE;
					MBATV0501E.control.auto_operate := TRUE;
					MBATV0501F.control.auto_operate := TRUE;
					MBAXV0519.control.auto_operate := TRUE;
					MBAXV0517.control.auto_operate := TRUE;
					MBATVT0510.control.auto_operate := TRUE;
					r08_add := FALSE;
					MBAS7_STEP[0].done := TRUE;
				END_IF;
			1:
				MBAXV0515.input.auto_open_signal := TRUE;
				MBAXV0518.input.auto_open_signal := TRUE;
				MBAXV0512.input.auto_open_signal := TRUE;
				MBAXV0524.input.auto_open_signal := TRUE;
				IF MBAXV0515.input.open_feedback_state AND MBAXV0518.input.open_feedback_state AND MBAXV0512.input.open_feedback_state AND MBAXV0524.input.open_feedback_state THEN
					MBAS7_STEP[1].done := TRUE;
				END_IF;
			2:
				CASE step7_2 OF
					0:
						IF NOT MBAS7_STEP[2].done THEN
							step7_2 := 1;
						END_IF;
					1:
						MBAXV0526.input.auto_open_signal := TRUE;
						step7_2 := 2;
					2:
						IF MBAPIT0501.status.value <= MBAS7_PARA_P1 THEN
							MBAXV0514.input.auto_open_signal := TRUE;
							IF MBAXV0514.input.open_feedback_state THEN
								step7_2 := 3;
							END_IF;
						END_IF;
					3:
						r08_add := TRUE;
						step7_2 := 0;
						MBAS7_STEP[2].done := TRUE;
				END_CASE;
			3:
				//观察R08进料视镜无液，反馈中控进料结束
			4:
				r08_add := FALSE;
				MBATV0501C.input.auto_open_signal := FALSE;
				IF MBATV0501C.input.close_feedback_state THEN
					MBATV0501E.input.auto_open_signal := FALSE;
				END_IF;
				MBATV0501F.input.auto_open_signal := TRUE;
				MBAXV0514.input.auto_open_signal := FALSE;
				MBAXV0512.input.auto_open_signal := FALSE;
				MBAXV0526.input.auto_open_signal := FALSE;
				//手动停R06
			5:
				CASE step7_5 OF
					0:
						IF NOT MBAS7_STEP[5].done THEN
							step7_5 := 1;
						END_IF;
					1:
						IF MBATIT0502.status.value <= MBAS7_PARA_Temp3 THEN
							MBAXV0519.input.auto_open_signal := TRUE;
							step7_5 := 2;
						END_IF;
					2:
						IF MBATIT0502.status.value <= MBAS7_PARA_Temp4 THEN
							MBAXV0519.input.auto_open_signal := FALSE;
							step7_5 := 3;
						END_IF;
					3:
						TON_5.PT := DINT_TO_TIME(MBAS7_PARA_T1 * 60 * 1000);
						TON_5.IN := TRUE;
						IF TON_5.Q THEN
							TON_5.IN := FALSE;
							step7_5 := 4;
						END_IF;
					4:
						MBAXV0518.input.auto_open_signal := FALSE;
						MBAXV0515.input.auto_open_signal := FALSE;
						MBAXV0517.input.auto_open_signal := FALSE;
						IF MBAXV0518.input.close_feedback_state AND MBAXV0515.input.close_feedback_state AND  MBAXV0517.input.close_feedback_state THEN
							step7_5 := 0;
							MBAS7_STEP[5].done := TRUE;
						END_IF;
				END_CASE;
				TON_5();
		END_CASE;
	END_IF;

	//转移物料控制温度压力
	IF r08_add THEN
		IF MBATIT0501.status.value >= MBAS7_PARA_Temp1 THEN
			MBATV0501F.input.auto_open_signal := TRUE;
			MBATV0501C.input.auto_open_signal := FALSE;
			MBATV0501E.input.auto_open_signal := FALSE;
		ELSIF MBATIT0501.status.value <= MBAS7_PARA_Temp2 THEN
			MBATV0501E.input.auto_open_signal := TRUE;
			MBATV0501F.input.auto_open_signal := FALSE;
			IF MBATV0501E.input.open_feedback_state THEN
				MBATV0501C.input.auto_open_signal := TRUE;
			END_IF;
		END_IF;
		IF MBAPIT0501.status.value >= MBAS7_PARA_P2 THEN
			MBAXV0526.input.auto_open_signal := TRUE;
		ELSIF MBAPIT0501.status.value <= MBAS7_PARA_P3 THEN
			MBAXV0526.input.auto_open_signal := FALSE;
		END_IF;
	END_IF;

	//TSV0510调节
	R_TRIG_1(CLK := MBATVT0510.status.auto_mode);
	IF R_TRIG_1.Q THEN
		MTBasicsPID_0.Enable := TRUE;
	END_IF;
	F_TRIG_1(CLK := MBATVT0510.status.auto_mode);
	IF F_TRIG_1.Q THEN
		MTBasicsPID_0.Enable := FALSE;
	END_IF;
	//MTBasicsPID_0.Enable := TRUE;
	MTBasicsPID_0.Invert := TRUE;
	MTBasicsPID_0.PIDParameters.Gain := MBAPid0510Para.gain;
	MTBasicsPID_0.PIDParameters.IntegrationTime := MBAPid0510Para.integration_time;
	MTBasicsPID_0.PIDParameters.DerivativeTime := MBAPid0510Para.derivative_time;
	MTBasicsPID_0.MinOut := 0.0;
	MTBasicsPID_0.MaxOut := 100.0;
	MTBasicsPID_0.SetValue := MBAPid0510Para.set_value;
	MTBasicsPID_0.ActValue := MBATIT0510.status.value;
	MTBasicsPID_0.Update := MBAPid0510.update;
	MTBasicsPID_0();
	MBAPid0510.out := MTBasicsPID_0.Out;
	IF MTBasicsPID_0.Active THEN
		MBATVT0510.input.auto_degree_set := MTBasicsPID_0.Out;
	ELSE
		MBATVT0510.input.auto_degree_set := 0.0;
	END_IF;
	IF MTBasicsPID_0.UpdateDone THEN
		MBAPid0510.update := FALSE;
	END_IF;

	//人工确认步骤可用
	IF (MBAS7.status.run_state) AND (NOT MBAS7_STEP[MBAS7.status.run_step].done AND ((MBAS7.status.run_step = 3) OR (MBAS7.status.run_step = 4))) THEN
		MBAS7.status.confirm_enable := TRUE;
	ELSE
		MBAS7.status.confirm_enable := FALSE;
	END_IF;
END_ACTION

(* ---- MBAS8_ACTION.st ---- *)
ACTION S8_ACT:
	//设定时间
	FOR i := 0 TO MBAS8_STEP_NUM DO
		IF MBAS8_ST[i] < T#5s THEN
			MBAS8_ST[i] := T#5s;
		END_IF;
		MBAS8_STEP[i].set_time := MBAS8_ST[i];
	END_FOR;

	//流程步骤
	ProcessHandleFC(MBAS8,MBAS8_STEP[0],MBAS8_STEP_NUM);

	//object 手自动切换
	IF (MBAS8.status.mode <> 0) AND (NOT MBAS8.auto_mode_edge) THEN
		MBAS8.auto_mode_edge := TRUE;
		MBAS8.manual_mode_edge := FALSE;

		MBAXV0516.control.auto_operate := TRUE;
		MBAXV0524.control.auto_operate := TRUE;
		MBAXV0520.control.auto_operate := TRUE;
		MBAXV0611.control.auto_operate := TRUE;
		MBAXV0603.control.auto_operate := TRUE;
		MBAXV0628.control.auto_operate := TRUE;
		MBAXV0613.control.auto_operate := TRUE;
		MBAPV0601.control.auto_operate := TRUE;
		MBAP06.control.auto_operate := TRUE;
		MBATV0601A.control.auto_operate := TRUE;
		MBATV0601B.control.auto_operate := TRUE;
		MBATV0601C.control.auto_operate := TRUE;
		MBATV0601D.control.auto_operate := TRUE;
		MBATV0601E.control.auto_operate := TRUE;
		MBATV0601F.control.auto_operate := TRUE;
		MBAXV0631.control.auto_operate := TRUE;
	END_IF;

	IF (MBAS8.status.mode = 0) AND (NOT MBAS8.manual_mode_edge) THEN
		MBAS8.manual_mode_edge := TRUE;
		MBAS8.auto_mode_edge := FALSE;

		MBAXV0516.control.manual_operate := TRUE;
		MBAXV0524.control.manual_operate := TRUE;
		MBAXV0520.control.manual_operate := TRUE;
		MBAXV0611.control.manual_operate := TRUE;
		MBAXV0603.control.manual_operate := TRUE;
		MBAXV0628.control.manual_operate := TRUE;
		MBAXV0613.control.manual_operate := TRUE;
		MBAPV0601.control.manual_operate := TRUE;
		MBAP06.control.manual_operate := TRUE;
		MBATV0601A.control.manual_operate := TRUE;
		MBATV0601B.control.manual_operate := TRUE;
		MBATV0601C.control.manual_operate := TRUE;
		MBATV0601D.control.manual_operate := TRUE;
		MBATV0601E.control.manual_operate := TRUE;
		MBATV0601F.control.manual_operate := TRUE;
		MBAXV0631.control.manual_operate := TRUE;
	END_IF;

	//错误信号停机
	MBAS8.input.error_signal := (MBAP06.status.motor_status >= 2) OR (MBAXV0516.status.valve_status >= 2) OR
	(MBAXV0524.status.valve_status >= 2) OR (MBAXV0520.status.valve_status >= 2) OR (MBAXV0611.status.valve_status >= 2) OR
	(MBAXV0603.status.valve_status >= 2) OR (MBAXV0628.status.valve_status >= 2) OR (MBAXV0613.status.valve_status >= 2) OR
	(MBAPV0601.status.valve_status >= 2) OR (MBATV0601A.status.valve_status >= 2) OR (MBATV0601B.status.valve_status >= 2) OR
	(MBATV0601C.status.valve_status >= 2) OR (MBATV0601D.status.valve_status >= 2) OR (MBATV0601E.status.valve_status >= 2) OR
	(MBATV0601F.status.valve_status >= 2) OR (MBAXV0631.status.valve_status >= 2);

	IF MBAS8.status.run_state = 1 THEN
		//步骤执行动作
		CASE MBAS8.status.run_step OF
			0:
				IF NOT MBAS8_STEP[0].done THEN
					MBAXV0516.control.auto_operate := TRUE;
					MBAXV0524.control.auto_operate := TRUE;
					MBAXV0520.control.auto_operate := TRUE;
					MBAXV0611.control.auto_operate := TRUE;
					MBAXV0603.control.auto_operate := TRUE;
					MBAXV0628.control.auto_operate := TRUE;
					MBAXV0613.control.auto_operate := TRUE;
					MBAPV0601.control.auto_operate := TRUE;
					MBAP06.control.auto_operate := TRUE;
					MBATV0601A.control.auto_operate := TRUE;
					MBATV0601B.control.auto_operate := TRUE;
					MBATV0601C.control.auto_operate := TRUE;
					MBATV0601D.control.auto_operate := TRUE;
					MBATV0601E.control.auto_operate := TRUE;
					MBATV0601F.control.auto_operate := TRUE;
					MBAXV0631.control.auto_operate := TRUE;
					is_press_ok_R09 := FALSE;
					MBAS8_STEP[0].done := TRUE;
				END_IF;
			1:
				//试漏
			2:
				//R09进料,人工观察R08转移完毕反馈
				CASE step8_2 OF
					0:
						IF NOT MBAS8_STEP[2].done THEN
							step8_2 := 1;
						END_IF;
					1:
						MBAXV0516.input.auto_open_signal := TRUE;
						IF MBAXV0516.input.open_feedback_state THEN
							step8_2 := 2;
						END_IF;
					2:
						IF MBAPIT0601.status.value <= MBAS8_PARA_P3 THEN
							MBAXV0524.input.auto_open_signal := FALSE;
							step8_2 := 3;
						END_IF;
					3:
						IF MBAXV0524.input.close_feedback_state THEN
							step8_2 := 4;
						END_IF;
					4:
						MBAXV0520.input.auto_open_signal := TRUE;
						MBAXV0611.input.auto_open_signal := TRUE;
						IF MBAXV0611.input.open_feedback_state THEN
							step8_2 := 5;
						END_IF;
					5:
						IF NOT MBAS8_STEP[2].done THEN
							IF MBAPIT0502.status.value <= MBAS8_PARA_P4 THEN
								MBAXV0520.input.auto_open_signal := TRUE;
							ELSIF MBAPIT0502.status.value >= MBAS8_PARA_P5 THEN
								MBAXV0520.input.auto_open_signal := FALSE;
							END_IF;
						ELSE
							step8_2 := 0;
						END_IF;
				END_CASE;
			3:
				MBAXV0520.input.auto_open_signal := FALSE;
				IF MBAPIT0502.status.value <= MBAS8_PARA_P6 THEN
					MBAXV0516.input.auto_open_signal := FALSE;
					MBAXV0524.input.auto_open_signal := TRUE;
					IF MBAXV0516.input.close_feedback_state AND MBAXV0524.input.open_feedback_state THEN
						MBAS8_STEP[3].done := TRUE;
					END_IF;
				END_IF;
			4:
				//吹扫 需人工观察
				IF NOT MBAS8_STEP[4].done THEN
					MBAXV0603.input.auto_open_signal := TRUE;
					IF MBAPIT0601.status.value >= MBAS8_PARA_P7 THEN
						MBAXV0611.input.auto_open_signal := TRUE;
					ELSIF MBAPIT0601.status.value <= MBAS8_PARA_P8 THEN
						MBAXV0611.input.auto_open_signal := FALSE;
					END_IF;
				ELSE
					MBAXV0603.input.auto_open_signal := FALSE;
					MBAXV0611.input.auto_open_signal := FALSE;
				END_IF;
			5:
				MBAXV0628.input.auto_open_signal := FALSE;
				MBAXV0613.input.auto_open_signal := TRUE;
				MBAPV0601.input.auto_open_signal := TRUE;
				//手动启动R09搅拌
			6:
				MBAP06.input.auto_run_signal := TRUE;
				IF MBAP06.input.run_feedback THEN
					MBAS8_STEP[6].done := TRUE;
				END_IF;
			7:
				HeatPot_4(ST1 := DINT_TO_TIME(MBAS8_PARA_T2 * 1000),
				ST2 := DINT_TO_TIME(MBAS8_PARA_T3 * 1000),
				V3 := MBATV0601E,
				V4 := MBATV0601F,
				V5 := MBATV0601C,
				V6 := MBATV0601D,
				done := MBAS8_STEP[7].done);
			8:
				IF MBATIT0601.status.value >= MBAS8_PARA_Temp1 THEN
					MBATV0601E.input.auto_open_signal := FALSE;
				END_IF;
			9:
				//降温
				MBATV0601E.input.auto_open_signal := FALSE;
				MBAXV0631.input.auto_open_signal := TRUE;
				CoolPot_2(
					time := cool_pot_time,
					V1 := MBATV0601A,
					V2 := MBATV0601B,
					V3 := MBATV0601D,
					V4 := MBATV0601F,
					V5 := MBATV0601C,
				done := MBAS8_STEP[9].done);
			10:
				CASE step8_10 OF
					0:
						IF NOT MBAS8_STEP[10].done THEN
							step8_10 := 1;
						END_IF;
					1:
						IF MBATIT0601.status.value <= MBAS8_PARA_Temp2 THEN
							MBAXV0631.input.auto_open_signal := FALSE;
							MBAXV0603.input.auto_open_signal := TRUE;
							step8_10 := 2;
						END_IF;
					2:
						IF MBAPIT0601.status.value >= MBAS8_PARA_P9 THEN
							MBAP06.input.auto_run_signal := FALSE;
							IF MBAP06.input.run_feedback = FALSE THEN
								step8_10 := 3;
							END_IF;
						END_IF;
					3:
						IF MBAPIT0601.status.value >= MBAS8_PARA_P10 THEN
							MBAXV0603.input.auto_open_signal := FALSE;
							step8_10 := 4;
						END_IF;
					4:
						MBAS8_STEP[10].done := TRUE;
						step8_10 := 0;
				END_CASE;
			11:
				MBAXV0628.input.auto_open_signal := TRUE;
				//				IF MBAXV0628.input.open_feedback_state THEN
				//					MBAS8_STEP[11].done := TRUE;
				//				END_IF;
			12:
				MBAXV0613.input.auto_open_signal := FALSE;
				MBATV0601A.input.auto_open_signal := FALSE;
				MBATV0601B.input.auto_open_signal := FALSE;
				IF MBAXV0613.input.close_feedback_state AND MBATV0601A.input.close_feedback_state AND MBATV0601B.input.close_feedback_state THEN
					MBAS8_STEP[12].done := TRUE;
				END_IF;
		END_CASE;
	END_IF;

	IF press_test_R09 THEN
		CASE step8_1 OF
			0:
				is_press_ok_R09 := FALSE;
				step8_1 := 1;
			1:
				MBAPV0601.input.auto_open_signal := FALSE;
				IF MBAPV0601.input.close_feedback_state THEN
					MBAXV0603.input.auto_open_signal := TRUE;
					step8_1 := 2;
				END_IF;
			2:
				IF MBAPIT0601.status.value >= MBAS8_PARA_P1 THEN
					MBAXV0603.input.auto_open_signal := FALSE;
					step8_1 := 3;
				END_IF;
			3:
				TON_12.PT := DINT_TO_TIME(MBAS8_PARA_T1 * 60 * 1000);
				TON_12.IN := TRUE;
				IF TON_12.Q THEN
					TON_12.IN := FALSE;
					step8_1 := 4;
				END_IF;
			4:
				IF MBAS8_PARA_P1 - MBAPIT0601.status.value <= MBAS8_PARA_P2 THEN
					is_press_ok_R09 := TRUE;
				ELSE
					is_press_ok_R09 := FALSE;
				END_IF;
				step8_1 := 5;
			5:
				press_test_R09 := FALSE;
				step8_1 := 0;
		END_CASE;
		TON_12();
	END_IF;

	//MBAR05酒精回收
	//常压回收
	IF r05_recover THEN
		CASE r05_recover_step OF
			0:
				MBAXV0616.control.auto_operate := TRUE;
				MBAFVT0601.control.auto_operate := TRUE;
				MBAR05.control.auto_operate := TRUE;
				MBATV0602E.control.auto_operate := TRUE;
				MBATV0602F.control.auto_operate := TRUE;
				MBATV0602C.control.auto_operate := TRUE;
				MBATV0602D.control.auto_operate := TRUE;
				MBATV0602A.control.auto_operate := TRUE;
				MBATV0602B.control.auto_operate := TRUE;
				r05_recover_step := 1;
			1:
				MBAXV0616.input.auto_open_signal := TRUE;
				MTBasicsPID_2.Enable := FALSE;
				MBAFVT0601.input.auto_degree_set := 0.0;
				MBAR05.input.auto_run_signal := TRUE;
				IF MBAXV0616.input.open_feedback_state AND MBAR05.input.auto_run_signal THEN
					r05_recover_step := 2;
				END_IF;
			2:
				HeatPot_1(ST1 := DINT_TO_TIME(MBAR05_PARA_T1 * 1000),
				ST2 := DINT_TO_TIME(MBAR05_PARA_T2 * 1000),
				V3 := MBATV0602E,
				V4 := MBATV0602F,
				V5 := MBATV0602C,
				V6 := MBATV0602D,
				done := HeatPot_1_done);
				IF HeatPot_1_done THEN
					HeatPot_1_done := FALSE;
					r05_recover_step := 3;
				END_IF;
			3:
				IF MBATIT0602.status.value >=  MBAR05_PARA_Temp1 THEN
					MBATV0602E.input.auto_open_signal := FALSE;
					r05_recover_step := 4;
				END_IF;
			4:
				TON_6.PT := DINT_TO_TIME(MBAR05_PARA_T3 * 60 * 1000);
				TON_6.IN := TRUE;
				IF TON_6.Q THEN
					TON_6.IN := FALSE;
					MTBasicsPID_2.Enable := TRUE;
					r05_recover_step := 5;
				END_IF;
			5:
				IF MBATIT0602.status.value >= MBAR05_PARA_Temp2 THEN
					MBATV0602F.input.auto_open_signal := FALSE;
					MBATV0602C.input.auto_open_signal := FALSE;
					MBATV0602D.input.auto_open_signal := TRUE;
					IF MBATV0602F.input.close_feedback_state AND MBATV0602C.input.close_feedback_state AND MBATV0602D.input.open_feedback_state THEN
						r05_recover_step := 6;
					END_IF;
				END_IF;
			6:
				TON_6.PT := DINT_TO_TIME(MBAR05_PARA_T4 * 1000);
				TON_6.IN := TRUE;
				IF TON_6.Q THEN
					TON_6.IN := FALSE;
					r05_recover_step := 7;
				END_IF;
			7:
				MBATV0602D.input.auto_open_signal := FALSE;
				IF MBATV0602D.input.close_feedback_state THEN
					MBATV0602A.input.auto_open_signal := TRUE;
				END_IF;
				IF MBATV0602A.input.open_feedback_state THEN
					MBATV0602B.input.auto_open_signal := TRUE;
				END_IF;
				IF MBATV0602A.input.open_feedback_state AND MBATV0602B.input.open_feedback_state AND MBATV0602D.input.close_feedback_state THEN
					r05_recover_step := 8;
				END_IF;
			8:
				IF MBATIT0602.status.value <= MBAR05_PARA_Temp3 THEN
					MTBasicsPID_2.Enable := FALSE;
					MBAFVT0601.input.auto_degree_set := 0.0;
					MBATV0602B.input.auto_open_signal := FALSE;
					IF MBATV0602B.input.close_feedback_state THEN
						MBATV0602A.input.auto_open_signal := FALSE;
						IF MBATV0602A.input.close_feedback_state THEN
							r05_recover_step := 9;
						END_IF;
					END_IF;
				END_IF;
			9:
				MBAR05.input.auto_run_signal := FALSE;
				MBAXV0616.input.auto_open_signal := FALSE;
				IF (NOT MBAR05.input.run_feedback) AND MBAXV0616.input.close_feedback_state THEN
					r05_recover_step := 0;
					r05_recover := FALSE;
				END_IF;
		END_CASE;
		TON_6();
	END_IF;

	//FVT0601 pid调节
	R_TRIG_2(CLK := MBAFVT0601.status.auto_mode);
	IF R_TRIG_2.Q THEN
		MTBasicsPID_2.Enable := TRUE;
	END_IF;
	F_TRIG_2(CLK := MBAFVT0601.status.auto_mode);
	IF F_TRIG_2.Q THEN
		MTBasicsPID_2.Enable := FALSE;
	END_IF;
	//MTBasicsPID_2.Enable := TRUE;
	MTBasicsPID_2.PIDParameters.Gain := MBAPidFVT0601Para.gain;
	MTBasicsPID_2.PIDParameters.IntegrationTime := MBAPidFVT0601Para.integration_time;
	MTBasicsPID_2.PIDParameters.DerivativeTime := MBAPidFVT0601Para.derivative_time;
	MTBasicsPID_2.MinOut := 0.0;
	MTBasicsPID_2.MaxOut := 100.0;
	MTBasicsPID_2.SetValue := MBAPidFVT0601Para.set_value;
	MTBasicsPID_2.ActValue := MBAFIT0601.flowrate;
	MTBasicsPID_2.Update := MBAPidFVT0601.update;
	MTBasicsPID_2();
	MBAPidFVT0601.out := MTBasicsPID_2.Out;
	IF MTBasicsPID_2.Active THEN
		MBAFVT0601.input.auto_degree_set := MTBasicsPID_2.Out + MBAPidFVT0601Para.min_out;
		//	ELSE
		//		MBAFVT0601.input.auto_degree_set := 0.0;
	END_IF;
	IF MTBasicsPID_2.UpdateDone THEN
		MBAPidFVT0601.update := FALSE;
	END_IF;

	//人工确认步骤可用
	IF (MBAS8.status.run_state) AND (NOT MBAS8_STEP[MBAS8.status.run_step].done AND ((MBAS8.status.run_step = 1) OR (MBAS8.status.run_step = 2) OR (MBAS8.status.run_step = 4) OR (MBAS8.status.run_step = 5) OR (MBAS8.status.run_step = 8) OR (MBAS8.status.run_step = 11))) THEN
		MBAS8.status.confirm_enable := TRUE;
	ELSE
		MBAS8.status.confirm_enable := FALSE;
	END_IF;
END_ACTION
